// TwinCAT 3 PLC project TAMAR2MM
// ProgramVersion: 3.1.4024.0
// libraries:
//   Tc2_MC2, * (Beckhoff Automation GmbH)
//   Tc2_Standard, * (Beckhoff Automation GmbH)
//   Tc2_System, * (Beckhoff Automation GmbH)
//   Tc2_Utilities, * (Beckhoff Automation GmbH)
//   Tc3_Module, * (Beckhoff Automation GmbH)
//   VisuDialogs, * (System)
// project tree:
//   / GlobalTextList.TcGTLO, PlcTask.TcTTO (not stored), Visualization Manager.TcVMO (not stored), VISU_TASK.TcTTO (not stored)
//   POUs/AXES/ AXES_CYCLE.TcPOU, FB_Axis.TcPOU, GVL_AXES.TcGVL (not stored), vAXIS.TcVIS, vAXIS_CONTROLLER.TcVIS, AXES_SCREEN.TcVIS
//   POUs/EVENT_LOGGER/ E_EventType.TcDUT, FB_EventLogger.TcPOU, GVL_EVENT_LOGGER.TcGVL, ST_Event.TcDUT, UpdateEventTimestampWithSystemTime.TcPOU (not stored), UpdateTimeStamp.TcPOU (not stored), vEVENT_LOGGER.TcVIS (not stored)
//   POUs/ E_STATE.TcDUT, GVL_MAIN.TcGVL, MACHINE.TcPOU, MAIN.TcPOU
//   POUs/IO/ EL1809.TcDUT, EL2809.TcDUT, GVL_IO.TcGVL, ST_VTUG.TcDUT
//   POUs/PISTONS/ E_PISTON_STATE.TcDUT, E_PISTON_TYPE.TcDUT, FB_PISTON.TcPOU, GVL_PISTONS.TcGVL, PIST_CYCLE.TcPOU, ST_PISTON.TcDUT (not stored), vPISTONS.TcVIS (not stored), vPISTON.TcVIS
//   POUs/STATIONS/ FB_FEEDER.TcPOU, FB_SEPARATE.TcPOU, FB_STATION.TcPOU, STATION_CYCLE.TcPOU, vFEEDER.TcVIS, vSEPARATE.TcVIS, vSTATION_CONTROLLER.TcVIS
//   VISUs/ vCOMM.TcVIS, vMACHINE.TcVIS
// real-time tasks:
//   TASK PlcTask: cycle T#10ms, priority 20, ADS port 350
//   TASK VISU_TASK: cycle T#200000us, priority 30, ADS port 351
// motion (NC):
//   TASK NC-Task 1 SAF: cycle T#2ms, priority 4, ADS port 501
//   TASK NC-Task 1 SVB: cycle T#10ms, priority 8, ADS port 511
//   AXIS MAIN_CONV (id 1)
//     OtherSettings: AllowMotionCmdToSlave=true
//     encoder EncType=1
//     drive DrvType=5
//       Analog: TorqueSetpointScale=10, ScaleFactorActTorque=0.1
//       TimeComp: TaskDelayCycles=1
//     controller CtrType=1
//       CtrPara: PriorControlFactor=1
//         Observer: BandWidth=20
//   AXIS SUP_CONV (id 2)
//     OtherSettings: AllowMotionCmdToSlave=true
//     encoder EncType=1
//     drive DrvType=5
//       Analog: TorqueSetpointScale=10, ScaleFactorActTorque=0.1
//       TimeComp: TaskDelayCycles=1
//     controller CtrType=1
//       CtrPara: PriorControlFactor=1
//         Observer: BandWidth=20
//   AXIS PRESS1A (id 3)
//     OtherSettings: AllowMotionCmdToSlave=true
//     encoder EncType=1
//     drive DrvType=5
//       Analog: TorqueSetpointScale=10, ScaleFactorActTorque=0.1
//       TimeComp: TaskDelayCycles=1
//     controller CtrType=1
//       CtrPara: PriorControlFactor=1
//         Observer: BandWidth=20
//   AXIS PRESS1B (id 4)
//     OtherSettings: AllowMotionCmdToSlave=true
//     encoder EncType=1
//     drive DrvType=5
//       Analog: TorqueSetpointScale=10, ScaleFactorActTorque=0.1
//       TimeComp: TaskDelayCycles=1
//     controller CtrType=1
//       CtrPara: PriorControlFactor=1
//         Observer: BandWidth=20
// variable links:
//   TAMAR2MM/TAMAR2MM Instance <-> NC-Task 1 SAF/Axes/MAIN_CONV
//     PlcTask Inputs/GVL_MAIN.MAIN_CONV.Axis.NcToPlc <-> Outputs/ToPlc
//     PlcTask Outputs/GVL_MAIN.MAIN_CONV.Axis.PlcToNc <-> Inputs/FromPlc
//   TAMAR2MM/TAMAR2MM Instance <-> NC-Task 1 SAF/Axes/SUP_CONV
//     PlcTask Inputs/GVL_MAIN.SUP_CONV.Axis.NcToPlc <-> Outputs/ToPlc
//     PlcTask Outputs/GVL_MAIN.SUP_CONV.Axis.PlcToNc <-> Inputs/FromPlc

// ---- POUs/EVENT_LOGGER/E_EventType.TcDUT
{attribute 'qualified_only'}
{attribute 'strict'}
TYPE E_EventType :
(
	Alarm := 0,
	Message:=1
);
END_TYPE

// ---- POUs/EVENT_LOGGER/ST_Event.TcDUT
TYPE ST_Event :
STRUCT
	eEventType: STRING(255); 
	eEventSeverity: STRING(255);
	nEventIdentity: UDINT;
	sEventName: STRING(255);
	sEventText: STRING(255);
	dtTimestamp: DATE_AND_TIME;
	
END_STRUCT
END_TYPE

// ---- POUs/E_STATE.TcDUT
{attribute 'qualified_only'}
{attribute 'strict'}
TYPE E_STATE :
(
	uninit:=0,
	ready,
	busy,
	error
	
);
END_TYPE

// ---- POUs/IO/EL1809.TcDUT
TYPE EL1809 :
STRUCT
	ch1		:BOOL;
	ch2		:BOOL;
	ch3		:BOOL;
	ch4		:BOOL;
	ch5		:BOOL;
	ch6		:BOOL;
	ch7		:BOOL;
	ch8		:BOOL;
	ch9		:BOOL;
	ch10		:BOOL;
	ch11		:BOOL;
	ch12		:BOOL;
	ch13		:BOOL;
	ch14		:BOOL;
	ch15		:BOOL;
	ch16		:BOOL;	
END_STRUCT
END_TYPE

// ---- POUs/IO/EL2809.TcDUT
TYPE EL2809 :
STRUCT
	ch1		:BOOL;
	ch2		:BOOL;
	ch3		:BOOL;
	ch4		:BOOL;
	ch5		:BOOL;
	ch6		:BOOL;
	ch7		:BOOL;
	ch8		:BOOL;
	ch9		:BOOL;
	ch10		:BOOL;
	ch11		:BOOL;
	ch12		:BOOL;
	ch13		:BOOL;
	ch14		:BOOL;
	ch15		:BOOL;
	ch16		:BOOL;	
END_STRUCT
END_TYPE

// ---- POUs/IO/ST_VTUG.TcDUT
TYPE ST_VTUG :
STRUCT
	sol_14: BOOL;
	sol_12: BOOL;
END_STRUCT
END_TYPE

// ---- POUs/PISTONS/E_PISTON_STATE.TcDUT
{attribute 'qualified_only'}
{attribute 'strict'}
TYPE E_PISTON_STATE :
(
	uninit:=0,
	ready,
	opening,
	opened,
	closing,
	closed,
	error,
	busy
);
END_TYPE

// ---- POUs/PISTONS/E_PISTON_TYPE.TcDUT
{attribute 'qualified_only'}
{attribute 'strict'}
TYPE E_PISTON_TYPE :
(
	NO_SENSORS,
	ONLY_OPEN,
	ONLY_CLOSE,
	BOTH
);
END_TYPE

// ---- POUs/EVENT_LOGGER/GVL_EVENT_LOGGER.TcGVL
//{attribute 'qualified_only'}
VAR_GLOBAL
	// ================================== error and logs ==============================
	sError:STRING;
	gEventType: STRING(255); 
	gEventSeverity: STRING(255);
	gEventIdentity: UDINT:=0;
	gEventText: STRING(255):='Startup Event';
	gEventName: STRING(255);
	sEventTime: STRING(255);
	fbEventLogger: FB_EventLogger;
	WriteLogToFile:BOOL:=FALSE;
	sLog:STRING(255);
	bBuffer_full:BOOL:=FALSE;
END_VAR

// ---- POUs/GVL_MAIN.TcGVL
//{attribute 'qualified_only'}
VAR_GLOBAL
	fbFEEDER: FB_FEEDER;
	fbSEPARATE1: FB_SEPARATE;
	fbSEPARATE2: FB_SEPARATE;
	MAIN_CONV:FB_Axis;
	SUP_CONV:FB_Axis;
	PRESS1A:FB_Axis;
	PRESS1B:FB_Axis;
	PIST1: FB_PISTON;
	PIST2: FB_PISTON;
	
	bMAIN_HOME:BOOL:=FALSE;
	bMAIN_HOMED:BOOL:=FALSE;
	sMAIN_STATE:STRING:='UNINIT';
	eMAIN_STATE: E_STATE:=E_STATE.uninit;
	bMAIN_RESET:BOOL:=FALSE;
	iMAIN_STATE: INT:=98;
	bMAIN_PAUSE:BOOL:=FALSE;
	bMAIN_START:BOOL:=FALSE;
	
END_VAR

// ---- POUs/IO/GVL_IO.TcGVL
//{attribute 'qualified_only'}
VAR_GLOBAL
	uIOLINK1 AT%Q* : ULINT;
	uIOLINK2 AT%Q* : ULINT;	

	inputs AT %I* : ARRAY [1..4] OF EL1809;
	outputs AT %Q* : ARRAY[1..1] OF EL2809;
	
	//manifold AT %Q* : ARRAY[1..3] OF ST_VTUG;

END_VAR

// ---- POUs/PISTONS/GVL_PISTONS.TcGVL
//{attribute 'qualified_only'}
VAR_GLOBAL
	
	pFEEDER_PUSH:  FB_PISTON;
	pFEEDER_HOLD1: FB_PISTON;
	pFEEDER_HOLD2: FB_PISTON;
	pFEEDER_OPEN1: FB_PISTON;
	pFEEDER_OPEN2: FB_PISTON;
	
	pSEPARATE1_LIFT:   FB_PISTON;
	pSEPARATE1_PUSH:   FB_PISTON;
	pSEPARATE1_COLET1: FB_PISTON;
	pSEPARATE1_COLET2: FB_PISTON;
	pSEPARATE1_COLET3: FB_PISTON;
	pSEPARATE1_COLET4: FB_PISTON;
	pSEPARATE1_JACK1:  FB_PISTON;
	pSEPARATE1_JACK2:  FB_PISTON;
	pSEPARATE1_JACK3:  FB_PISTON;
	pSEPARATE1_JACK4:  FB_PISTON;
	pSEPARATE1_DRAWR:  FB_PISTON;
	pSEPARATE1_PINS1:  FB_PISTON;
	pSEPARATE1_PINS2:  FB_PISTON;
	
	pSEPARATE2_PUSH:   FB_PISTON;
	pSEPARATE2_LIFT:   FB_PISTON;
	pSEPARATE2_COLET1: FB_PISTON;
	pSEPARATE2_COLET2: FB_PISTON;
	pSEPARATE2_COLET3: FB_PISTON;
	pSEPARATE2_COLET4: FB_PISTON;
	pSEPARATE2_JACK1:  FB_PISTON;
	pSEPARATE2_JACK2:  FB_PISTON;
	pSEPARATE2_JACK3:  FB_PISTON;
	pSEPARATE2_JACK4:  FB_PISTON;
	pSEPARATE2_DRAWR:  FB_PISTON;
	pSEPARATE2_PINS1:  FB_PISTON;
	pSEPARATE2_PINS2:  FB_PISTON;
	
	
	
END_VAR

// ---- POUs/EVENT_LOGGER/FB_EventLogger.TcPOU
FUNCTION_BLOCK FB_EventLogger
VAR_INPUT
END_VAR
VAR_OUTPUT
END_VAR
VAR
	buffer_counter:INT;
	EventBuffer: ARRAY[1..MAXIMUN_SIZE_OF_EVENT_BUFFR] OF ST_Event;
	EventBuffer_clear: ARRAY[1..MAXIMUN_SIZE_OF_EVENT_BUFFR] OF ST_Event;
	EventBufferIndex:INT:=0;
END_VAR
VAR CONSTANT
	MAXIMUN_SIZE_OF_EVENT_BUFFR:INT :=100;
END_VAR

METHOD IsEventBufferFull : BOOL
VAR_INPUT
END_VAR
IF (EventBufferIndex+1) > MAXIMUN_SIZE_OF_EVENT_BUFFR THEN
	EventBuffer:=EventBuffer_clear;
	EventBufferIndex:=0 ;
	//IsEventBufferFull:=TRUE; 
END_IF
IsEventBufferFull:=FALSE;
END_METHOD

(* returns false if not succesfull*) 
METHOD PUBLIC mAdd : BOOL
VAR_INPUT
	
END_VAR

VAR
	arrDataToWrite: INT;
END_VAR

IF NOT IsEventBufferFull() THEN
	EventBufferIndex:=EventBufferIndex+1;
	EventBuffer[EventBufferIndex].eEventType:=gEventType;
	EventBuffer[EventBufferIndex].eEventSeverity:=gEventSeverity;
	EventBuffer[EventBufferIndex].nEventIdentity:=gEventIdentity;
	EventBuffer[EventBufferIndex].sEventName:=gEventName;
	EventBuffer[EventBufferIndex].sEventText:=gEventText;
	UpdateEventTimestampWithSystemTime (stEvent:=EventBuffer[EventBufferIndex]); 
	sEventTime:= DT_TO_STRING (EventBuffer[EventBufferIndex].dtTimestamp);
	mAdd:=TRUE ;
ELSE
	mAdd:=FALSE;
END_IF
END_METHOD

END_FUNCTION_BLOCK

// ---- POUs/STATIONS/FB_FEEDER.TcPOU
FUNCTION_BLOCK FB_FEEDER EXTENDS FB_STATION
VAR_INPUT
	fbPUSH: REFERENCE TO FB_PISTON;
	fbHOLD1: REFERENCE TO FB_PISTON;
	fbHOLD2: REFERENCE TO FB_PISTON;
	fbOPEN1: REFERENCE TO FB_PISTON;
	fbOPEN2: REFERENCE TO FB_PISTON;
	rACTION_TIME: TIME;
	bTEST:BOOL;
END_VAR
VAR_OUTPUT
END_VAR
VAR
	bSTART_ACTION:BOOL;
	
END_VAR

tACTION(IN:= bSTART_ACTION, PT:=rACTION_TIME , Q=> , ET=> );
IF bRESET THEN
	bRESET:=FALSE;
	iSTATION_STATE:=98 ;
	bPAUSE:=FALSE;
END_IF

IF iSTATION_STATE<>98 AND (fbHOLD1.eSTATE= E_STATE.error OR fbHOLD2.eSTATE= E_STATE.error OR fbOPEN1.eSTATE= E_STATE.error OR fbOPEN2.eSTATE= E_STATE.error OR fbPUSH.eSTATE= E_STATE.error)  THEN 
	iSTATION_STATE:=99;
END_IF

CASE iSTATION_STATE OF 
	1:
		bHOME:=FALSE;
		iSTATION_STATE:=100;
		bHOMED:=TRUE;
	2: //open open hold
		bSTART:=FALSE;
		eSTATE:=E_STATE.busy;
		sSTATION_STATE:='HOLD AND OPEN';
		fbHOLD1.aOPEN();
		fbHOLD2.aOPEN();
		fbOPEN1.aOPEN();
		fbOPEN2.aOPEN();
		IF fbHOLD1.eSTATE= E_STATE.busy AND fbHOLD2.eSTATE= E_STATE.busy AND fbOPEN1.eSTATE= E_STATE.busy AND fbOPEN2.eSTATE= E_STATE.busy  THEN
			iSTATION_STATE:=3;
		END_IF
	3://wait fo open and hold and then push
		IF  fbHOLD1.eSTATE= E_STATE.ready AND fbHOLD2.eSTATE= E_STATE.ready AND fbOPEN1.eSTATE= E_STATE.ready AND fbOPEN2.eSTATE= E_STATE.ready THEN
			IF NOT bPAUSE THEN
				sSTATION_STATE:='OPEN PUSH';
				fbPUSH.aOPEN();
				IF fbPUSH.eSTATE= E_STATE.busy THEN
					iSTATION_STATE:=4;
				END_IF
			END_IF
		END_IF
	4:	//wait for push and close push
		IF fbPUSH.eSTATE= E_STATE.ready THEN
			IF NOT bPAUSE THEN
				sSTATION_STATE:='CLOSE PUSH';
				fbPUSH.aCLOSE();
				IF fbPUSH.eSTATE= E_STATE.busy THEN
					iSTATION_STATE:=5;
				END_IF
			END_IF
		END_IF
	5://wait for push close and close hold and open
		IF fbPUSH.eSTATE= E_STATE.ready THEN
			IF NOT bPAUSE THEN
				sSTATION_STATE:='RELEASE AND CLOSE';
				fbHOLD1.aCLOSE();
				fbHOLD2.aCLOSE();
				fbOPEN1.aCLOSE();
				fbOPEN2.aCLOSE();
				IF fbPUSH.eSTATE= E_STATE.ready AND fbHOLD1.eSTATE= E_STATE.ready AND fbHOLD2.eSTATE= E_STATE.ready AND fbOPEN1.eSTATE= E_STATE.ready AND fbOPEN2.eSTATE= E_STATE.ready THEN
					 iSTATION_STATE:=6;
				END_IF
			END_IF
		END_IF

	6:	//open pist 3
		IF fbPUSH.eSTATE= E_STATE.ready AND fbHOLD1.eSTATE= E_STATE.ready AND fbHOLD2.eSTATE= E_STATE.ready AND fbOPEN1.eSTATE= E_STATE.ready AND fbOPEN2.eSTATE= E_STATE.ready THEN
			iSTATION_STATE:=100;
		END_IF
	
	
	98:
		bHOMED:=FALSE;
		eSTATE:=E_STATE.uninit;
		sSTATION_STATE:='UNINIT';
		bRESET:=FALSE;
		fbPUSH.aRESET();
		fbHOLD1.aRESET();
		fbHOLD2.aRESET();
		fbOPEN1.aRESET();
		fbOPEN2.aRESET();
		IF fbPUSH.eSTATE= E_STATE.uninit AND fbHOLD1.eSTATE= E_STATE.uninit AND fbHOLD2.eSTATE= E_STATE.uninit AND fbOPEN1.eSTATE= E_STATE.uninit AND fbOPEN2.eSTATE= E_STATE.uninit THEN
			iSTATION_STATE:=980;
		END_IF
	980: 
		IF fbPUSH.eSTATE= E_STATE.ready AND fbHOLD1.eSTATE= E_STATE.ready AND fbHOLD2.eSTATE= E_STATE.ready AND fbOPEN1.eSTATE= E_STATE.ready AND fbOPEN2.eSTATE= E_STATE.ready THEN
			IF bHOME THEN
				iSTATION_STATE:=1;
			END_IF
		END_IF
		
		//IF fbPIST1.bERROR OR fbPIST2.bERROR OR fbPIST3.bERROR THEN
		//	iSTATION_STATE:=99;
	//	END_IF
	
	99:
		eSTATE:=E_STATE.error;
		sSTATION_STATE:='PISTON ERROR';
		
	100:
		eSTATE:=E_STATE.ready;
		sSTATION_STATE:='READY';
		IF bSTART THEN
			bSTART:=FALSE;
			iSTATION_STATE:=2;
		END_IF
		
END_CASE

END_FUNCTION_BLOCK

// ---- POUs/STATIONS/FB_STATION.TcPOU
FUNCTION_BLOCK FB_STATION
VAR_INPUT
	eSTATE:E_STATE:=E_STATE.uninit;
	sSTATION_STATE:STRING:='UNINIT';
	sName:STRING;
	bHOMED : BOOL:=FALSE;
	tACTION:TON;
	bPAUSE:BOOL:=FALSE;
	bHOME: BOOL:=FALSE;
	
	
END_VAR
VAR_OUTPUT
END_VAR
VAR
	bERROR:BOOL;
	bRESET:BOOL;
	bSTART:BOOL:=FALSE;
	iSTATION_STATE:INT:=98;;
	bFIRST_RUN:BOOL:=FALSE;
END_VAR

ACTION aHOME:
bHOME:=TRUE;
END_ACTION

ACTION aRESET:
bRESET:=TRUE;
END_ACTION

ACTION aSTART:
bSTART:=TRUE;
END_ACTION

END_FUNCTION_BLOCK

// ---- POUs/PISTONS/FB_PISTON.TcPOU
FUNCTION_BLOCK FB_PISTON
VAR_INPUT
	eSTATE:E_STATE:=E_STATE.uninit;
	sSTATE:STRING:='UNINIT';
	sNAME:STRING;
	bLOCAL_MANUAL: BOOL:=FALSE;
	pist_TYPE: E_PISTON_TYPE;
	pist_STATE: E_PISTON_STATE:=E_PISTON_STATE.uninit;
	rOPEN_TIME: TIME;
	rCLOSE_TIME: TIME;
	rOPEN_TIMEOUT: TIME;
	tCLOSE_TIMEOUT: TIME;
	bOPEN_LIMIT: BOOL;
	bCLOSED_LIMIT: BOOL;
	bOPEN_CMD: BOOL;
	bCLOSE_CMD: BOOL;
	bOPEN_SWR: BOOL;
	bCLOSE_SWR: BOOL;
	bCONDITION: BOOL:=TRUE;
	bLOCAL_RESET:BOOL;
	bOPEN_DEFAULT: BOOL;
	
END_VAR
VAR_OUTPUT
	bOPEN_VALVE: BOOL;
	bCLOSE_VALVE: BOOL;
	bBUSY:BOOL;
	bOPENED:BOOL;
	bCLOSED:BOOL;
	bERROR:BOOL:=FALSE;
END_VAR
VAR
	T_OPEN: TON;
	T_OPEN_TIMEOUT: TON;
	T_CLOSE: TON;
	T_CLOSE_TIMEOUT: TON;
	
	bFIRST_DONE: BOOL:=FALSE;
	
END_VAR

T_OPEN(IN:= bOPEN_CMD, PT:=rOPEN_TIME , Q=> , ET=> );
T_CLOSE(IN:=  NOT bOPEN_CMD, PT:=rCLOSE_TIME , Q=> , ET=> );
T_OPEN_TIMEOUT(IN:= bOPEN_CMD , PT:= rOPEN_TIMEOUT, Q=> , ET=> );
T_CLOSE_TIMEOUT(IN:=  NOT bOPEN_CMD , PT:= tCLOSE_TIMEOUT, Q=> , ET=> );

IF bLOCAL_RESET THEN//========================== RESET================
	bLOCAL_RESET:=FALSE;
	pist_STATE:=E_PISTON_STATE.uninit;
END_IF

IF NOT bLOCAL_MANUAL THEN//====================== MANUAL ==============
	bOPEN_CMD:=bOPEN_SWR;
END_IF

IF NOT bFIRST_DONE THEN  // ============== check default mode ===============
	bFIRST_DONE:=TRUE;
	bOPEN_CMD:=bOPEN_DEFAULT;
END_IF
//================================================== UNINIT =====================================================
CASE pist_STATE OF
	E_PISTON_STATE.uninit:
		eSTATE:=E_STATE.uninit;
		bOPEN_CMD:=bOPEN_DEFAULT;
		bOPEN_SWR:=bOPEN_DEFAULT;
		bERROR:=FALSE;
		IF bOPEN_CMD  THEN
			bOPEN_VALVE:=TRUE;
			bCLOSE_VALVE:=FALSE;
			pist_STATE:=E_PISTON_STATE.opening;
		ELSE
			bOPEN_VALVE:=FALSE;
			bCLOSE_VALVE:=TRUE;
			pist_STATE:=E_PISTON_STATE.closing;
		END_IF
//================================================== OPENING =====================================================
	E_PISTON_STATE.opening:
	eSTATE:=E_STATE.busy;
	sSTATE:='OPENING';
	bBUSY:=TRUE; bOPENED:=FALSE; bCLOSED:=FALSE;
	CASE pist_TYPE OF//------------------------------no sensors
		E_PISTON_TYPE.NO_SENSORS:
		IF T_OPEN.Q THEN
			pist_STATE:=E_PISTON_STATE.opened;
		END_IF
		//----------------------------- both sensors
		E_PISTON_TYPE.BOTH:
		IF bOPEN_LIMIT THEN
			pist_STATE:=E_PISTON_STATE.opened;
		END_IF
		IF T_OPEN_TIMEOUT.Q THEN
			bOPEN_CMD:=FALSE;
			aPISTON_ERROR();
			pist_STATE:=E_PISTON_STATE.error;
		END_IF
		//----------------------------- only open sensor
		E_PISTON_TYPE.ONLY_OPEN:
		IF bOPEN_LIMIT THEN
			pist_STATE:=E_PISTON_STATE.opened;
		END_IF
		IF T_OPEN_TIMEOUT.Q THEN
			bOPEN_CMD:=FALSE;
			aPISTON_ERROR();
			pist_STATE:=E_PISTON_STATE.error;
		END_IF
		//----------------------------- only close sensor
		E_PISTON_TYPE.ONLY_CLOSE:
		IF T_OPEN.Q THEN
			pist_STATE:=E_PISTON_STATE.opened;
		END_IF
	END_CASE
//================================================== CLOSING =====================================================	
	E_PISTON_STATE.closing:
	eSTATE:=E_STATE.busy;
	sSTATE:='CLOSING'; bOPENED:=FALSE; bCLOSED:=FALSE;
	bBUSY:=TRUE;
	CASE pist_TYPE OF//--------------------------------------- no sensors
		E_PISTON_TYPE.NO_SENSORS:
		IF T_CLOSE.Q THEN
			pist_STATE:=E_PISTON_STATE.closed;
		END_IF
		//-------------------------------------- both sensors
		E_PISTON_TYPE.BOTH:
		IF bCLOSED_LIMIT THEN
			pist_STATE:=E_PISTON_STATE.closed;
		END_IF
		IF T_CLOSE_TIMEOUT.Q THEN
			bOPEN_CMD:=TRUE;
			pist_STATE:=E_PISTON_STATE.error;
		END_IF
		//-------------------------------------- only close sensor
		E_PISTON_TYPE.ONLY_CLOSE:
		IF bCLOSED_LIMIT THEN
			pist_STATE:=E_PISTON_STATE.closed;
		END_IF
		IF T_CLOSE_TIMEOUT.Q THEN
			bOPEN_CMD:=TRUE;
			aPISTON_ERROR();
			pist_STATE:=E_PISTON_STATE.error;
		END_IF
		//----------------------------- only close sensor
		E_PISTON_TYPE.ONLY_OPEN:
		IF T_CLOSE.Q THEN
			pist_STATE:=E_PISTON_STATE.closed;
		END_IF
	END_CASE
//================================================== OPENED =====================================================	
	E_PISTON_STATE.opened:
	eSTATE:=E_STATE.ready;
	sSTATE:='OPENED';
	bBUSY:=FALSE; bOPENED:=TRUE; bCLOSED:=FALSE;
	IF NOT bOPEN_CMD  THEN
		pist_STATE:=E_PISTON_STATE.closing;
		bOPEN_VALVE:=FALSE;
		bCLOSE_VALVE:=TRUE;
	END_IF
	CASE pist_TYPE OF
		//-------------------------------------- both sensors
		E_PISTON_TYPE.BOTH:
		IF NOT bOPEN_LIMIT THEN
			bOPEN_CMD:=FALSE;
			aPISTON_ERROR();
			pist_STATE:=E_PISTON_STATE.error;
		END_IF
		//-------------------------------------- only open sensor
		E_PISTON_TYPE.ONLY_OPEN:
		IF NOT bOPEN_LIMIT THEN
			bOPEN_CMD:=FALSE;
			aPISTON_ERROR();
			pist_STATE:=E_PISTON_STATE.error;
		END_IF
	END_CASE
//================================================== CLOSED =====================================================	
	E_PISTON_STATE.closed:
	eSTATE:=E_STATE.ready;
	sSTATE:='CLOSED';
	bBUSY:=FALSE; bOPENED:=FALSE; bCLOSED:=TRUE;
	IF bOPEN_CMD  THEN
		pist_STATE:=E_PISTON_STATE.opening;
		bOPEN_VALVE:=TRUE;
		bCLOSE_VALVE:=FALSE;
	END_IF
	CASE pist_TYPE OF
		//-------------------------------------- both sensors
		E_PISTON_TYPE.BOTH:
		IF NOT bCLOSED_LIMIT THEN
			bOPEN_CMD:=TRUE;
			aPISTON_ERROR();
			pist_STATE:=E_PISTON_STATE.error;
		END_IF
		//-------------------------------------- only close sensor
		E_PISTON_TYPE.ONLY_CLOSE:
		IF NOT bCLOSED_LIMIT THEN
			bOPEN_CMD:=TRUE;
			aPISTON_ERROR();
			pist_STATE:=E_PISTON_STATE.error;
		END_IF
	END_CASE
//================================================== ERROR =====================================================	
	E_PISTON_STATE.error:
		eSTATE:=E_STATE.error;
		sSTATE:='ERROR';
		bERROR:=TRUE;
	//
END_CASE

ACTION aCLOSE:
bOPEN_SWR:=FALSE;
END_ACTION

ACTION aHOME:
IF bOPEN_DEFAULT THEN
	bOPEN_SWR:=TRUE;
ELSE
	bOPEN_SWR:=FALSE;
END_IF
END_ACTION

ACTION aOPEN:
bOPEN_SWR:=TRUE;
END_ACTION

ACTION aPISTON_ERROR:
gEventType:= 'piston Alarm'; 
gEventSeverity:= 'Error';

gEventName:= sNAME;
IF pist_STATE=E_PISTON_STATE.opening  THEN
	gEventText:='piston opening';
	gEventIdentity:=1001;
END_IF
IF pist_STATE=E_PISTON_STATE.closing THEN
	gEventText:='piston closing';
	gEventIdentity:=1002;
END_IF
IF pist_STATE=E_PISTON_STATE.closed THEN
	gEventText:='piston closed';
	gEventIdentity:=1003;
END_IF
IF pist_STATE=E_PISTON_STATE.opened THEN
	gEventText:='piston opened';
	gEventIdentity:=1004;
END_IF
fbEventLogger.mAdd();
END_ACTION

ACTION aRESET:
bLOCAL_RESET:=TRUE;
END_ACTION

END_FUNCTION_BLOCK

// ---- POUs/STATIONS/FB_SEPARATE.TcPOU
FUNCTION_BLOCK FB_SEPARATE  EXTENDS FB_STATION
VAR_INPUT
	fbPUSH:   REFERENCE TO FB_PISTON;
	fbLIFT:   REFERENCE TO FB_PISTON;
	fbCOLET1: REFERENCE TO FB_PISTON;
	fbCOLET2: REFERENCE TO FB_PISTON;
	fbCOLET3: REFERENCE TO FB_PISTON;
	fbCOLET4: REFERENCE TO FB_PISTON;
	fbJACK1:  REFERENCE TO FB_PISTON;
	fbJACK2:  REFERENCE TO FB_PISTON;
	fbJACK3:  REFERENCE TO FB_PISTON;
	fbJACK4:  REFERENCE TO FB_PISTON;
	fbDRAWR:  REFERENCE TO FB_PISTON;
	fbPINS1:  REFERENCE TO FB_PISTON;
	fbPINS2:  REFERENCE TO FB_PISTON;
	fbPRESS1A:REFERENCE TO FB_Axis;
	fbPRESS1B:REFERENCE TO FB_Axis;
	
END_VAR
VAR_OUTPUT
END_VAR
VAR
END_VAR

IF bRESET THEN
	bRESET:=FALSE;
	iSTATION_STATE:=98 ;
	bPAUSE:=FALSE;
END_IF

IF iSTATION_STATE<>98 AND (fbLIFT.eSTATE= E_STATE.error OR
							 fbCOLET1.eSTATE= E_STATE.error OR 
								fbCOLET2.eSTATE= E_STATE.error OR
									fbCOLET3.eSTATE= E_STATE.error OR 
										fbCOLET4.eSTATE= E_STATE.error OR
											fbJACK1.eSTATE= E_STATE.error OR
												 fbJACK2.eSTATE= E_STATE.error OR 
													fbJACK3.eSTATE= E_STATE.error OR
														fbJACK4.eSTATE= E_STATE.error OR 
															fbDRAWR.eSTATE= E_STATE.error OR
																fbPINS1.eSTATE= E_STATE.error OR
												 					fbPINS2.eSTATE= E_STATE.error OR
																		fbPUSH.eSTATE= E_STATE.error  )THEN									
																										 
	iSTATION_STATE:=99;
END_IF

CASE iSTATION_STATE OF 
	1: //open pist 1
		bSTART:=FALSE;
		eSTATE:=E_STATE.busy;
		sSTATION_STATE:='LIFT DOWN';
		fbLIFT.aOPEN();
		IF fbLIFT.eSTATE= E_STATE.busy THEN
			iSTATION_STATE:=2;
		END_IF
	2://wait for LIFT ready
		IF fbLIFT.eSTATE= E_STATE.ready THEN
			IF NOT bPAUSE THEN
				iSTATION_STATE:=3;
			END_IF
		END_IF
	3:	//CLOSE COLET 1 2  ======================================= SEPARATE A =====================
		sSTATION_STATE:='CLOSE COLET 1 2';
		fbCOLET1.aOPEN();
		fbCOLET2.aOPEN();
		IF fbCOLET1.eSTATE= E_STATE.busy AND fbCOLET2.eSTATE= E_STATE.busy THEN
			iSTATION_STATE:=4;
		END_IF
	4:// WAIT FOR COLET 1 2
		IF fbCOLET1.eSTATE= E_STATE.ready AND fbCOLET2.eSTATE= E_STATE.ready THEN
			IF NOT bPAUSE THEN
				iSTATION_STATE:=5;
			END_IF
		END_IF
	5:	//SEPARATE A 
		sSTATION_STATE:='SEPARATE A';
		fbLIFT.aCLOSE();
		fbPRESS1A.mMOVE_REL(1000);
		fbPRESS1B.mMOVE_REL(1000);
		
		IF fbLIFT.eSTATE= E_STATE.busy AND fbPRESS1A.eSTATE= E_STATE.busy AND fbPRESS1B.eSTATE= E_STATE.busy THEN
			iSTATION_STATE:=6;
		END_IF
	6:
		IF  fbPRESS1A.eSTATE= E_STATE.ready AND fbPRESS1B.eSTATE= E_STATE.ready THEN
			IF NOT bPAUSE THEN
				iSTATION_STATE:=7;
			END_IF
		END_IF
		
	7:	//CLOSE COLET 1 2  ======================================= SEPARATE B =====================
		sSTATION_STATE:='CLOSE COLET 3 4';
		fbCOLET3.aOPEN();
		fbCOLET4.aOPEN();
		IF fbCOLET3.eSTATE= E_STATE.busy AND fbCOLET4.eSTATE= E_STATE.busy THEN
			iSTATION_STATE:=8;
		END_IF
	8:// WAIT FOR COLET 1 2
		IF fbCOLET3.eSTATE= E_STATE.ready AND fbCOLET4.eSTATE= E_STATE.ready THEN
			IF NOT bPAUSE THEN
				iSTATION_STATE:=9;
			END_IF
		END_IF
	9:	//SEPARATE A 
		sSTATION_STATE:='SEPARATE B';
		fbPRESS1A.mMOVE_REL(1000);
		fbPRESS1B.mMOVE_REL(1000);
		
		IF fbPRESS1A.eSTATE= E_STATE.busy AND fbPRESS1B.eSTATE= E_STATE.busy THEN
			iSTATION_STATE:=10;
		END_IF
	10:
		IF  fbLIFT.eSTATE= E_STATE.ready AND fbPRESS1A.eSTATE= E_STATE.ready AND fbPRESS1B.eSTATE= E_STATE.ready THEN
			IF NOT bPAUSE THEN
				iSTATION_STATE:=11;
			END_IF
		END_IF
		
		//========================================================================== CLEARING =======================
	11:	
		sSTATION_STATE:='OPEN DRAWER';
		fbDRAWR.aOPEN();
		IF fbDRAWR.eSTATE= E_STATE.busy  THEN
			iSTATION_STATE:=12;
		END_IF
	12:
		IF fbDRAWR.eSTATE= E_STATE.ready THEN
			IF NOT bPAUSE THEN
				iSTATION_STATE:=13;
			END_IF
		END_IF
	13:	//open colets
		sSTATION_STATE:='OPEN COLETS';
		fbCOLET1.aCLOSE();
		fbCOLET2.aCLOSE();
		fbCOLET3.aCLOSE();
		fbCOLET4.aCLOSE();
		IF fbCOLET1.eSTATE= E_STATE.busy AND fbCOLET2.eSTATE= E_STATE.busy AND fbCOLET3.eSTATE= E_STATE.busy AND fbCOLET4.eSTATE= E_STATE.busy THEN
			iSTATION_STATE:=14;
		END_IF
	14:
		IF fbCOLET1.eSTATE= E_STATE.ready AND fbCOLET2.eSTATE= E_STATE.ready AND fbCOLET3.eSTATE= E_STATE.ready AND fbCOLET4.eSTATE= E_STATE.ready THEN
			IF NOT bPAUSE THEN
				iSTATION_STATE:=15;
			END_IF
		END_IF	
	15:	//press pins
		sSTATION_STATE:='PINS OUT';
		fbPINS1.aOPEN();
		fbPINS2.aOPEN();
		IF fbPINS1.eSTATE= E_STATE.busy AND fbPINS2.eSTATE= E_STATE.busy THEN
			iSTATION_STATE:=16;
		END_IF
	16:
		IF fbPINS1.eSTATE= E_STATE.ready AND fbPINS2.eSTATE= E_STATE.ready THEN
			IF NOT bPAUSE THEN
				iSTATION_STATE:=17;
			END_IF
		END_IF
	17:	//pins up and push
		sSTATION_STATE:='PINS UP AND PUSH';
		fbPINS1.aCLOSE();
		fbPINS2.aCLOSE();
		fbPUSH.aOPEN();
		IF fbPUSH.eSTATE= E_STATE.busy AND fbPINS1.eSTATE= E_STATE.busy AND fbPINS2.eSTATE= E_STATE.busy THEN
			iSTATION_STATE:=18;
		END_IF
	18:
		IF  fbPUSH.eSTATE= E_STATE.ready AND fbPINS1.eSTATE= E_STATE.ready AND fbPINS2.eSTATE= E_STATE.ready THEN
			IF NOT bPAUSE THEN
				iSTATION_STATE:=19;
			END_IF
		END_IF
	19:	//close drawer jacks down
		sSTATION_STATE:='CLOSE DRAWER JACKS DOWN';
		fbDRAWR.aCLOSE();
		fbPRESS1A.aHOME();
		fbPRESS1B.aHOME();
		IF fbDRAWR.eSTATE= E_STATE.busy AND fbPRESS1A.eSTATE= E_STATE.busy AND fbPRESS1B.eSTATE= E_STATE.busy THEN
			iSTATION_STATE:=20;
		END_IF
	20:
		IF  fbLIFT.eSTATE= E_STATE.ready AND fbDRAWR.eSTATE= E_STATE.ready AND fbPRESS1A.bHOME AND fbPRESS1B.bHOMED THEN
			IF NOT bPAUSE THEN
				iSTATION_STATE:=100;
			END_IF
		END_IF

	
	98:
		eSTATE:=E_STATE.uninit;
		sSTATION_STATE:='UNINIT';
		bRESET:=FALSE;
		fbPRESS1A.aHOME();
		fbPRESS1B.aHOME();
		fbPUSH.aRESET();
		fbLIFT.aRESET();
		fbCOLET1.aRESET();
		fbCOLET2.aRESET();
		fbCOLET3.aRESET();
		fbCOLET4.aRESET();
		fbJACK1.aRESET();
		fbJACK2.aRESET();
		fbJACK3.aRESET();
		fbJACK4.aRESET();
		fbDRAWR.aRESET();
		fbPINS1.aRESET();
		fbPINS2.aRESET();
		
		IF fbPRESS1A.eSTATE= E_STATE.busy AND 
					fbPRESS1B.eSTATE= E_STATE.busy AND 
						fbLIFT.eSTATE= E_STATE.uninit AND
							 fbCOLET1.eSTATE= E_STATE.uninit AND
								fbCOLET2.eSTATE= E_STATE.uninit AND
									fbCOLET3.eSTATE= E_STATE.uninit AND
										fbCOLET4.eSTATE= E_STATE.uninit AND
											fbJACK1.eSTATE= E_STATE.uninit AND
												 fbJACK2.eSTATE= E_STATE.uninit AND 
													fbJACK3.eSTATE= E_STATE.uninit AND
														fbJACK4.eSTATE= E_STATE.uninit AND 
															fbDRAWR.eSTATE= E_STATE.uninit AND
																fbPINS1.eSTATE= E_STATE.uninit AND
												 					fbPINS2.eSTATE= E_STATE.uninit AND
																		fbPUSH.eSTATE= E_STATE.uninit THEN
			iSTATION_STATE:=980;
		END_IF
	980: 
		IF fbPRESS1A.bHOMED AND 
				fbPRESS1B.bHOMED AND 
					fbLIFT.eSTATE= E_STATE.ready AND
						 fbCOLET1.eSTATE= E_STATE.ready AND
							fbCOLET2.eSTATE= E_STATE.ready AND
								fbCOLET3.eSTATE= E_STATE.ready AND
									fbCOLET4.eSTATE= E_STATE.ready AND
										fbJACK1.eSTATE= E_STATE.ready AND
											fbJACK2.eSTATE= E_STATE.ready AND 
												fbJACK3.eSTATE= E_STATE.ready AND
													fbJACK4.eSTATE= E_STATE.ready AND 
														fbDRAWR.eSTATE= E_STATE.ready AND
															fbPINS1.eSTATE= E_STATE.ready AND
																fbPINS2.eSTATE= E_STATE.ready AND
																	fbPUSH.eSTATE= E_STATE.ready THEN
			iSTATION_STATE:=100;
		END_IF
		
	
	99:
		eSTATE:=E_STATE.error;
		sSTATION_STATE:='ERROR';
		
	100:
		eSTATE:=E_STATE.ready;
		sSTATION_STATE:='READY';
		IF bSTART THEN
			bSTART:=FALSE;
			iSTATION_STATE:=1;
		END_IF
		
END_CASE

END_FUNCTION_BLOCK

// ---- POUs/AXES/FB_Axis.TcPOU
FUNCTION_BLOCK FB_Axis
VAR_INPUT
	eSTATE:E_STATE:=E_STATE.uninit;
	sAXIS_STATE:STRING:='UNINIT';
	sName:STRING;
	Axis:Axis_ref;
	bEnable:BOOL:=FALSE;
	bHalt:BOOL:=FALSE;
	bHOME:BOOL:=FALSE;
	bHOME_DIR:BOOL;
	bReset:BOOL:=FALSE;
	bSetPosition:BOOL:=FALSE;
	Dist:REAL;
	bMoveRel:BOOL:=FALSE;
	bMoveRelBusy:BOOL;
	rPos:LREAL;
	rVel:LREAL;
	rAcc:LREAL;
	rDec:LREAL;
	rJerk:LREAL;
	bMoveABS:BOOL:=FALSE;
	bMoveAbsBusy:BOOL;
	bJogPos:BOOL;
	bJogNeg:BOOL;
	bMANUAL:BOOL:=FALSE;
	tACTION:TON;
	ton_Reset: TON;
	bOPEN:BOOL;
	bCLOSE:BOOL;
	bLIMIT_OPENED:BOOL;
	bLIMIT_CLOSED:BOOL;
	bLIMIT:BOOL;
	rACTION_TIMEOUT:TIME:=T#10S;
	jogVEL: REAL;
	bSTOP:BOOL;
	SKIP_HOME :BOOL:=TRUE;
END_VAR

VAR_OUTPUT
	bOPENED:BOOL;
	bCLOSED:BOOL;
	bHOMED:BOOL;
	bBusy: BOOL;
	bAXIS_ERROR:BOOL;
	bSTATE_ERROR:BOOL;
	bInPos:BOOL;
	rActPos:LREAL;
	rActVel:LREAL;
	bRelDone:BOOL;
	bAbsDone:BOOL;
	bHaltDone:BOOL;
END_VAR
VAR
	bSTART_ACTION:BOOL;
	iHOME_STATE: INT:=98;
	iAXIS_STATE:INT:=98;
	tDelay: TON;
	bDelay:BOOL:=FALSE;
	MoveAbsolute: MC_MoveAbsolute;
	power: MC_Power;
	Reset: MC_Reset;
	SetPosition: MC_SetPosition;
	JOG: MC_Jog;
	RELATIVE: MC_MoveRelative;
	HALT: MC_Halt;
	HOME: MC_Home;
	bFirst_run:BOOL:=FALSE;
	bStopBusy:BOOL;
	
	
	
	
END_VAR

IF NOT bFirst_run THEN
	RESET.Execute:=TRUE;
	 bFirst_run:=TRUE;
END_IF

rActPos:=Axis.NcToPlc.ActPos;
rActVel:=Axis.NcToPlc.ActVelo;

IF RELATIVE.Done AND bMoveRel THEN
	bMoveRel:=FALSE;
END_IF

IF MoveAbsolute.Done AND bMoveAbs THEN
	bMoveAbs:=FALSE;
END_IF

IF RELATIVE.Busy OR JOG.Busy OR moveAbsolute.busy  THEN
	bBusy:=TRUE;
	//bInpos:=FALSE;
END_IF

IF NOT RELATIVE.Busy AND NOT JOG.Busy AND NOT moveAbsolute.busy  THEN
	bBusy:=FALSE;
	//bInpos:=TRUE;
END_IF

IF POWER.error OR RELATIVE.error OR MoveAbsolute.error OR JOG.error THEN
	bAXIS_ERROR:=TRUE;
END_IF


IF bRelDone OR  bAbsDone THEN
	bInPos:=TRUE;
END_IF


IF bBusy THEN
	bInPos:=FALSE;
	bRelDone:=FALSE;
	bAbsDone:=FALSE;
END_IF


CMDs();
mAXIS_STATE_MACHINE();

ACTION aAXIS_ERROR:
gEventType:= 'axis Alarm'; 
gEventSeverity:= 'Error';

gEventName:= sNAME;
IF iAXIS_STATE=1  THEN
	gEventText:='axis homing';
	gEventIdentity:=2001;
END_IF
IF iAXIS_STATE=20  THEN
	gEventText:='axis opening';
	gEventIdentity:=2002;
END_IF
IF iAXIS_STATE=40  THEN
	gEventText:='axis closing';
	gEventIdentity:=2003;
END_IF
fbEventLogger.mAdd();
END_ACTION

ACTION aHOME:
bHOME:=TRUE;
END_ACTION

ACTION aRESET:
iAXIS_STATE:=98;
bHOME:=FALSE;
END_ACTION

METHOD clear_cmd_req : BOOL
VAR_INPUT
END_VAR

bMoveABS:= bMoveRel:= bJogPos:= bJogNeg:=FALSE;
END_METHOD

ACTION CMDs:
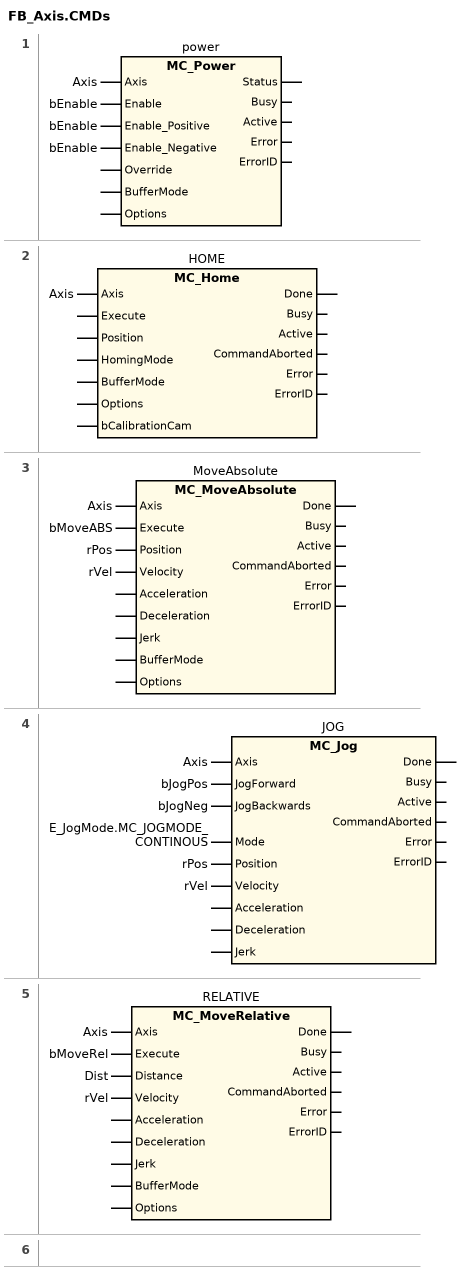
// NETWORK 1
power(Axis := Axis, Enable := bEnable, Enable_Positive := bEnable, Enable_Negative := bEnable); // MC_Power

// NETWORK 2
HOME(Axis := Axis); // MC_Home

// NETWORK 3
MoveAbsolute(Axis := Axis, Execute := bMoveABS, Position := rPos, Velocity := rVel); // MC_MoveAbsolute

// NETWORK 4
JOG(
    Axis := Axis,
    JogForward := bJogPos,
    JogBackwards := bJogNeg,
    Mode := E_JogMode.MC_JOGMODE_CONTINOUS,
    Position := rPos,
    Velocity := rVel); // MC_Jog

// NETWORK 5
RELATIVE(Axis := Axis, Execute := bMoveRel, Distance := Dist, Velocity := rVel); // MC_MoveRelative

// NETWORK 6

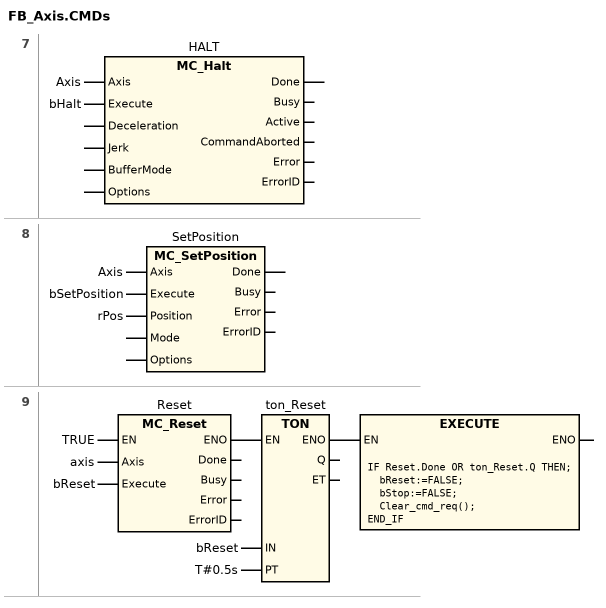
// NETWORK 7
HALT(Axis := Axis, Execute := bHalt); // MC_Halt

// NETWORK 8
SetPosition(Axis := Axis, Execute := bSetPosition, Position := rPos); // MC_SetPosition

// NETWORK 9
Reset(Axis := axis, Execute := bReset); // MC_Reset
ton_Reset(IN := bReset, PT := T#0.5s); // TON

IF Reset.Done OR ton_Reset.Q THEN;
	bReset:=FALSE;
	bStop:=FALSE;
	Clear_cmd_req();
END_IF
END_ACTION

METHOD mAXIS_STATE_MACHINE : BOOL
VAR_INPUT
	
END_VAR
tACTION(IN:= bSTART_ACTION, PT:=rACTION_TIMEOUT , Q=> , ET=> );
IF bHOME_DIR THEN
	bLIMIT:=bLIMIT_OPENED;
ELSE
	bLIMIT:=bLIMIT_CLOSED;
END_IF


CASE iAXIS_STATE OF
	1:// ============================================== HOMING
		bENABLE:=TRUE;
		bHOME:=FALSE;
		IF SKIP_HOME THEN
			bHOMED:=TRUE;
			IF bHOME_DIR THEN
				iAXIS_STATE:=100;// to ready state
			ELSE
				iAXIS_STATE:=100;// to ready state
			END_IF
		ELSE
			eSTATE:=E_STATE.busy;
			bSTART_ACTION:=TRUE;
			sAXIS_STATE:='HOMING - TO SENSOR';
			bHOMED:=FALSE;bHOME:=FALSE;
			bENABLE:=TRUE;
			rVel:= jogVEL;
			IF bHOME_DIR THEN
				bJogPos:=TRUE;
			ELSE
				bJogNeg:=TRUE;
			END_IF
			
			IF bLIMIT THEN
				bSTART_ACTION:=FALSE;
				bJogNeg:=FALSE;
				bJogPos:=FALSE;
				iAXIS_STATE:=2;
			END_IF
			IF tACTION.Q THEN
				bSTART_ACTION:=FALSE;
				aAXIS_ERROR();
				iAXIS_STATE:=99;
				bSTATE_ERROR:=TRUE;
			END_IF
		END_IF
		
	2://FROM LIMIT
			sAXIS_STATE:= 'HOMING- FROM SENSOR';
			IF Axis.NcToPlc.ActVelo= 0 THEN
				rVel:= jogVEL/5;
				IF bHOME_DIR THEN
					bJogNeg:=TRUE;
				ELSE
					bJogPos:=TRUE;
				END_IF
				iAXIS_STATE:=3;
			END_IF	
	3:// FINISH
			IF NOT bLIMIT THEN
				bJogNeg:=FALSE;
				bJogPos:=FALSE;
				IF Axis.NcToPlc.ActVelo= 0 THEN
					bHOMED:=TRUE;
					IF bHOME_DIR THEN
						iAXIS_STATE:=100;// to ready state
					ELSE
						iAXIS_STATE:=100;// to ready state
					END_IF
				END_IF
			END_IF
	
	50:	//========================ABSOLUTE=====================
	eSTATE:=E_STATE.busy;
	sAXIS_STATE:='MOVING ABSOLUTE';
	bAbsDone:=FALSE; bHOMED:=FALSE;bHOME:=FALSE;
	IF moveAbsolute.Done OR HALT.Done THEN
		iAXIS_STATE:=100;
		bAbsDone:=TRUE;
		bMoveAbs:=FALSE;
	END_IF
	51://========================RELATIVE=====================
	eSTATE:=E_STATE.busy;
	sAXIS_STATE:='MOVING RELATIVE';
	bRelDone:=FALSE;bHOMED:=FALSE;bHOME:=FALSE;
	IF RELATIVE.Done OR HALT.Done THEN
		iAXIS_STATE:=100; 
		bRelDone:=TRUE;
		bMoveRel:=FALSE;
	END_IF
	52://======================= HALT =========================
	sAXIS_STATE:='HALTING';
	bHaltDone:=FALSE;bHOMED:=FALSE;bHOME:=FALSE;
	IF HALT.Done THEN
		iAXIS_STATE:=100;
		bHaltDone:=TRUE;
		bHALT:=FALSE;
	END_IF		
	98:// ====================== UNINIT =========================
		eSTATE:=E_STATE.uninit;
		sAXIS_STATE:='UNINIT';
		bENABLE:=FALSE;
		bHOMED:=FALSE;
		IF bHOME THEN
			iAXIS_STATE:=1;
			bSTATE_ERROR:=FALSE;
		END_IF
		
	99://====================== ERROR ============================
		eSTATE:=E_STATE.error;
		sAXIS_STATE:='AXIS STATE ERROR';
		bJogNeg:=FALSE;
		bJogPos:=FALSE;
		bHOMED:=FALSE;
		IF bHOME THEN
			iAXIS_STATE:=1;
			bSTATE_ERROR:=FALSE;
		END_IF
		
	100://==================== READY =============================
		eSTATE:=E_STATE.ready;
		sAXIS_STATE:='READY';
		IF bHOME AND NOT bHOMED THEN
			iAXIS_STATE:=1;
			//bSTATE_ERROR:=FALSE;
		END_IF
		IF bCLOSE AND NOT bCLOSED THEN
			iAXIS_STATE:=40;
			bSTATE_ERROR:=FALSE;
		END_IF
		IF bOPEN AND NOT bOPENED THEN
			iAXIS_STATE:=20;
			bSTATE_ERROR:=FALSE;
		END_IF
		IF bMoveAbs THEN
			bENABLE:=TRUE;
			iAXIS_STATE:=50;
			bSTATE_ERROR:=FALSE;
		END_IF
		IF bMoveRel THEN
			bENABLE:=TRUE;
			iAXIS_STATE:=51;
			bSTATE_ERROR:=FALSE;
		END_IF
		IF bHALT THEN
			iAXIS_STATE:=52;
			bSTATE_ERROR:=FALSE;
		END_IF
	
END_CASE
END_METHOD

METHOD mMOVE_ABS : BOOL
VAR_INPUT
	movement:REAL;
END_VAR
rPOS:=movement;
bMoveAbs:=TRUE;
END_METHOD

METHOD mMOVE_REL : BOOL
VAR_INPUT
	movement:REAL;
END_VAR

IF eSTATE= E_STATE.ready THEN
	Dist:=movement;
	bMoveRel:=TRUE;
END_IF
END_METHOD

END_FUNCTION_BLOCK

// ---- POUs/AXES/AXES_CYCLE.TcPOU
PROGRAM AXES_CYCLE
VAR
END_VAR

GRP1();

ACTION GRP1:
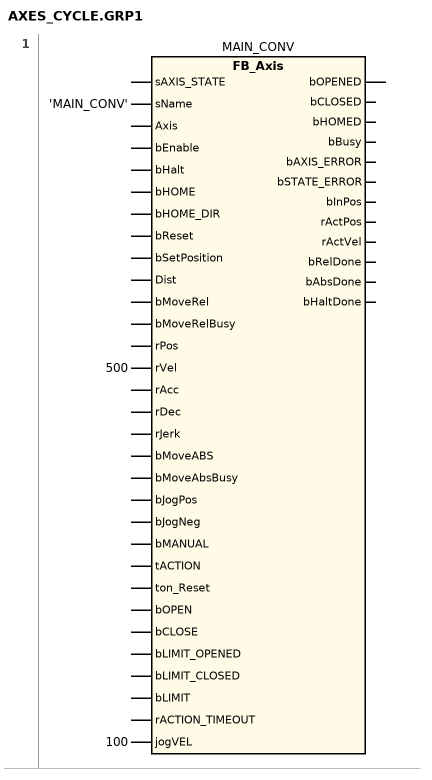
// NETWORK 1
MAIN_CONV(sName := 'MAIN_CONV', rVel := 500, jogVEL := 100); // FB_Axis

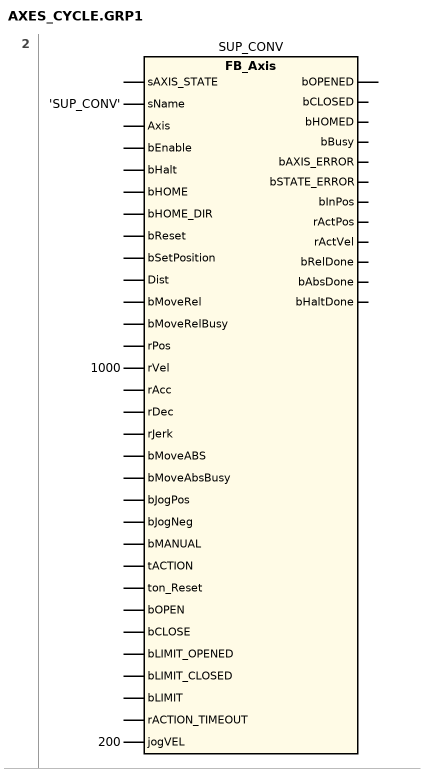
// NETWORK 2
SUP_CONV(sName := 'SUP_CONV', rVel := 1000, jogVEL := 200); // FB_Axis

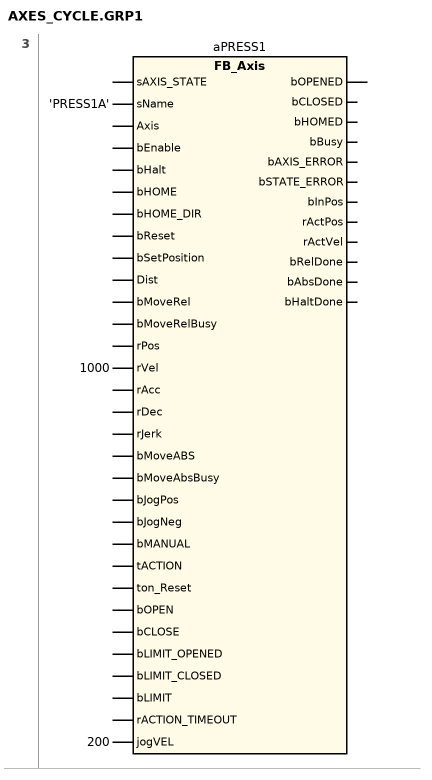
// NETWORK 3
aPRESS1(sName := 'PRESS1A', rVel := 1000, jogVEL := 200); // FB_Axis

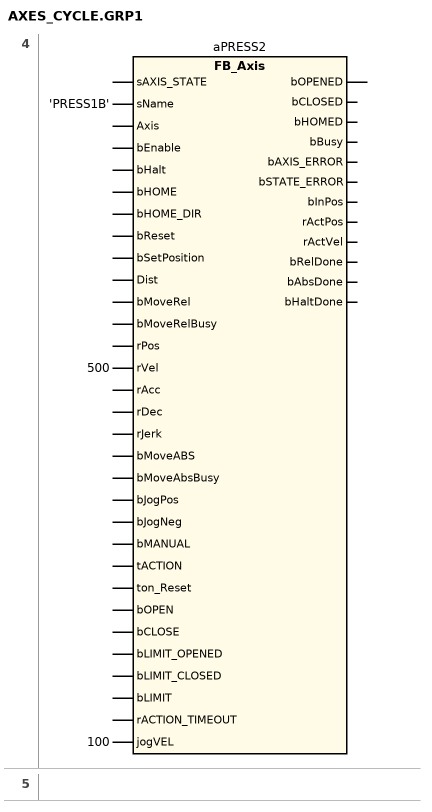
// NETWORK 4
aPRESS2(sName := 'PRESS1B', rVel := 500, jogVEL := 100); // FB_Axis

// NETWORK 5
END_ACTION

END_PROGRAM

// ---- POUs/MACHINE.TcPOU
PROGRAM MACHINE
VAR
END_VAR

IF fbFEEDER.eSTATE= E_STATE.error OR fbSEPARATE1.eSTATE= E_STATE.error OR MAIN_CONV.eSTATE= E_STATE.error OR SUP_CONV.eSTATE= E_STATE.error THEN
	iMAIN_STATE:=99 ;
END_IF

IF bMAIN_RESET THEN
	iMAIN_STATE:=98 ;
	bMAIN_PAUSE:=FALSE;
	sMAIN_STATE:='UNINIT';
END_IF

CASE iMAIN_STATE OF 
	1://===================================== HOME ============================
		MAIN_CONV.aHOME();
		SUP_CONV.aHOME();
		
		eMAIN_STATE:=E_STATE.busy;
		bMAIN_HOME:=FALSE;
		sMAIN_STATE:='HOMING';
		IF MAIN_CONV.bHOMED AND SUP_CONV.bHOMED THEN
			iMAIN_STATE:=100;
			bMAIN_HOMED:=TRUE;
		END_IF
	2: //====================================  START ==============================
		eMAIN_STATE:=E_STATE.busy;
		sMAIN_STATE:='CONVAYORS';
		MAIN_CONV.mMOVE_REL(1000);
		SUP_CONV.mMOVE_REL(1000);
		IF SUP_CONV.eSTATE= E_STATE.busy AND MAIN_CONV.eSTATE = E_STATE.busy THEN
			iMAIN_STATE:=3;
		END_IF
	3://wait for convayors
		IF SUP_CONV.eSTATE= E_STATE.ready AND MAIN_CONV.eSTATE = E_STATE.ready THEN
			IF NOT bMAIN_PAUSE THEN
				iMAIN_STATE:=4;
			END_IF
		END_IF
		
	4: //stations
		eMAIN_STATE:=E_STATE.busy;
		sMAIN_STATE:=' STANIONS';
		fbFEEDER.aSTART();
		fbSEPARATE1.aSTART();
		fbSEPARATE2.aSTART();
		IF fbSEPARATE1.eSTATE= E_STATE.busy AND fbSEPARATE2.eSTATE= E_STATE.busy AND fbFEEDER.eSTATE= E_STATE.busy THEN
			iMAIN_STATE:=5;
		END_IF
	5://wait for separate1
		IF fbSEPARATE1.eSTATE= E_STATE.ready AND fbSEPARATE2.eSTATE= E_STATE.ready AND fbFEEDER.eSTATE= E_STATE.ready THEN
			IF NOT bMAIN_PAUSE THEN
				iMAIN_STATE:=100;
			END_IF
		END_IF
		
	98://======================================== UNINIT ============================
		bMAIN_HOMED:=FALSE;
		eMAIN_STATE:=E_STATE.uninit;
		sMAIN_STATE:='UNINIT';
		bMAIN_RESET:=FALSE;
		fbFEEDER.aRESET();
		fbSEPARATE1.aRESET();
		MAIN_CONV.aRESET();
		
		IF fbFEEDER.eSTATE = E_STATE.uninit AND fbSEPARATE1.eSTATE = E_STATE.uninit AND MAIN_CONV.eSTATE=E_STATE.uninit  AND SUP_CONV.eSTATE=E_STATE.uninit THEN
			iMAIN_STATE:=980;
		END_IF
	980: 
		IF fbFEEDER.eSTATE= E_STATE.ready AND fbSEPARATE1.eSTATE= E_STATE.ready AND MAIN_CONV.eSTATE=E_STATE.uninit  AND SUP_CONV.eSTATE=E_STATE.uninit THEN
			IF bMAIN_HOME THEN
				iMAIN_STATE:=1;
			END_IF
		END_IF
	
	99://========================================== ERROR ================================
		eMAIN_STATE:=E_STATE.error;
		sMAIN_STATE:='MACHINE ERROR';
		
	100://========================================= READY ================================
		eMAIN_STATE:=E_STATE.ready;
		sMAIN_STATE:='READY';
		IF bMAIN_START THEN
			bMAIN_START:=FALSE;
			iMAIN_STATE:=2;
		END_IF
		
END_CASE

END_PROGRAM

// ---- POUs/MAIN.TcPOU
PROGRAM MAIN
VAR
	
END_VAR



AXES_CYCLE();
PIST_CYCLE();
STATION_CYCLE();
MACHINE();

END_PROGRAM

// ---- POUs/PISTONS/PIST_CYCLE.TcPOU
PROGRAM PIST_CYCLE
VAR
	bFirstRun:BOOL:=FALSE;
	counter :INT;
END_VAR


grp_feeder();
grp_separate1();
grp_separate2();

ACTION grp_feeder:
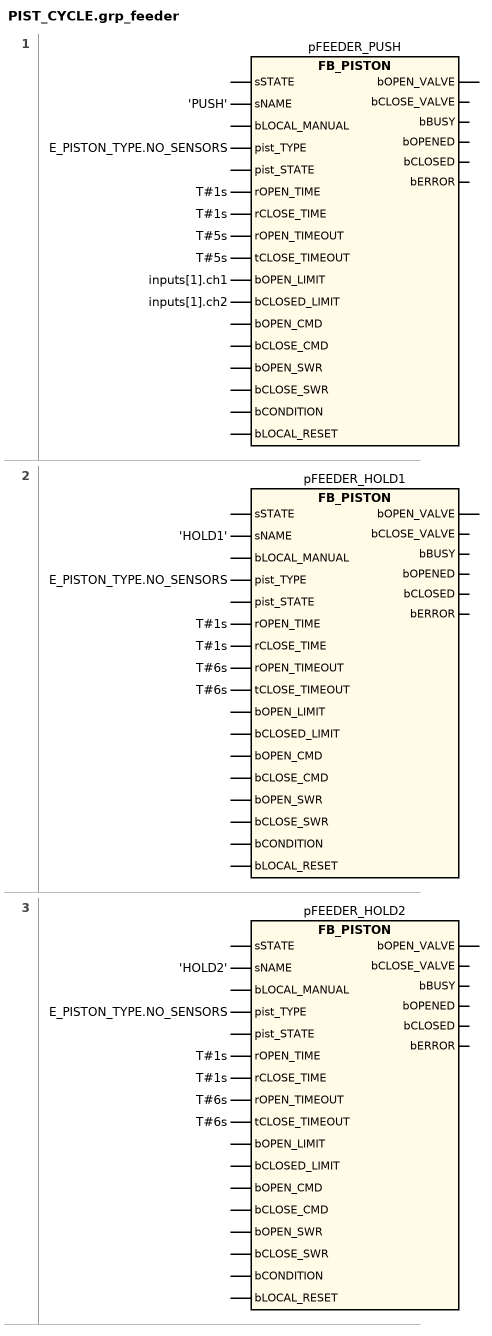
// NETWORK 1
pFEEDER_PUSH(
    sNAME := 'PUSH',
    pist_TYPE := E_PISTON_TYPE.NO_SENSORS,
    rOPEN_TIME := T#1s,
    rCLOSE_TIME := T#1s,
    rOPEN_TIMEOUT := T#5s,
    tCLOSE_TIMEOUT := T#5s,
    bOPEN_LIMIT := inputs[1].ch1,
    bCLOSED_LIMIT := inputs[1].ch2); // FB_PISTON

// NETWORK 2
pFEEDER_HOLD1(
    sNAME := 'HOLD1',
    pist_TYPE := E_PISTON_TYPE.NO_SENSORS,
    rOPEN_TIME := T#1s,
    rCLOSE_TIME := T#1s,
    rOPEN_TIMEOUT := T#6s,
    tCLOSE_TIMEOUT := T#6s); // FB_PISTON

// NETWORK 3
pFEEDER_HOLD2(
    sNAME := 'HOLD2',
    pist_TYPE := E_PISTON_TYPE.NO_SENSORS,
    rOPEN_TIME := T#1s,
    rCLOSE_TIME := T#1s,
    rOPEN_TIMEOUT := T#6s,
    tCLOSE_TIMEOUT := T#6s); // FB_PISTON

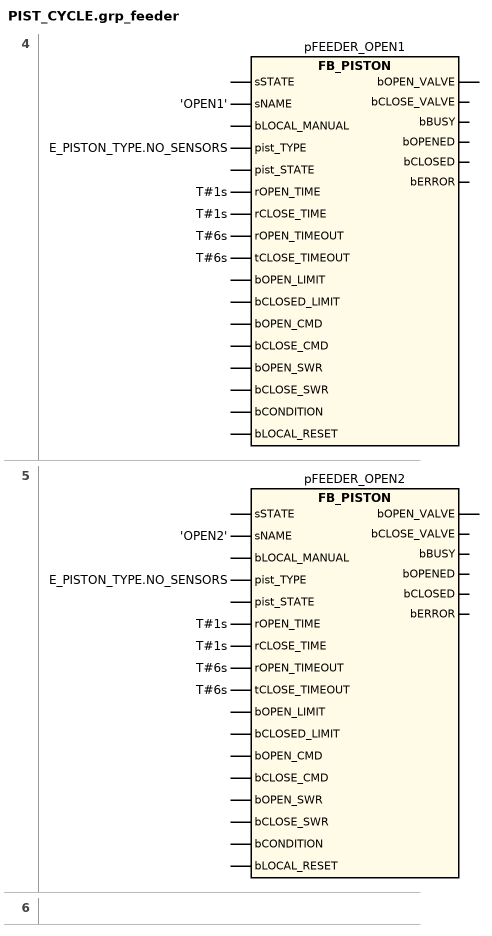
// NETWORK 4
pFEEDER_OPEN1(
    sNAME := 'OPEN1',
    pist_TYPE := E_PISTON_TYPE.NO_SENSORS,
    rOPEN_TIME := T#1s,
    rCLOSE_TIME := T#1s,
    rOPEN_TIMEOUT := T#6s,
    tCLOSE_TIMEOUT := T#6s); // FB_PISTON

// NETWORK 5
pFEEDER_OPEN2(
    sNAME := 'OPEN2',
    pist_TYPE := E_PISTON_TYPE.NO_SENSORS,
    rOPEN_TIME := T#1s,
    rCLOSE_TIME := T#1s,
    rOPEN_TIMEOUT := T#6s,
    tCLOSE_TIMEOUT := T#6s); // FB_PISTON

// NETWORK 6
END_ACTION

ACTION grp_separate1:
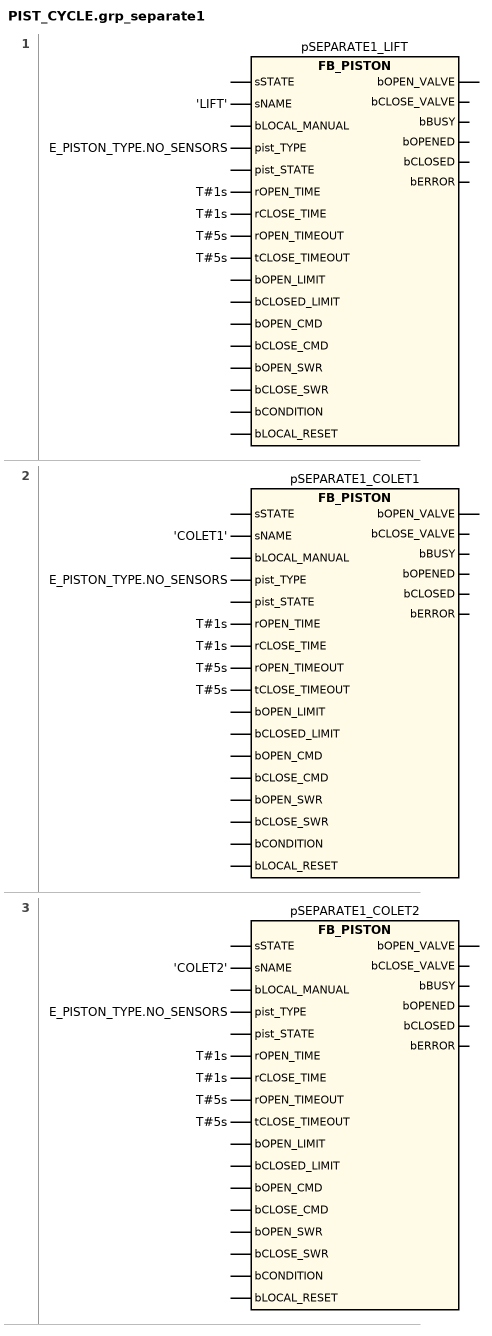
// NETWORK 1
pSEPARATE1_LIFT(
    sNAME := 'LIFT',
    pist_TYPE := E_PISTON_TYPE.NO_SENSORS,
    rOPEN_TIME := T#1s,
    rCLOSE_TIME := T#1s,
    rOPEN_TIMEOUT := T#5s,
    tCLOSE_TIMEOUT := T#5s); // FB_PISTON

// NETWORK 2
pSEPARATE1_COLET1(
    sNAME := 'COLET1',
    pist_TYPE := E_PISTON_TYPE.NO_SENSORS,
    rOPEN_TIME := T#1s,
    rCLOSE_TIME := T#1s,
    rOPEN_TIMEOUT := T#5s,
    tCLOSE_TIMEOUT := T#5s); // FB_PISTON

// NETWORK 3
pSEPARATE1_COLET2(
    sNAME := 'COLET2',
    pist_TYPE := E_PISTON_TYPE.NO_SENSORS,
    rOPEN_TIME := T#1s,
    rCLOSE_TIME := T#1s,
    rOPEN_TIMEOUT := T#5s,
    tCLOSE_TIMEOUT := T#5s); // FB_PISTON

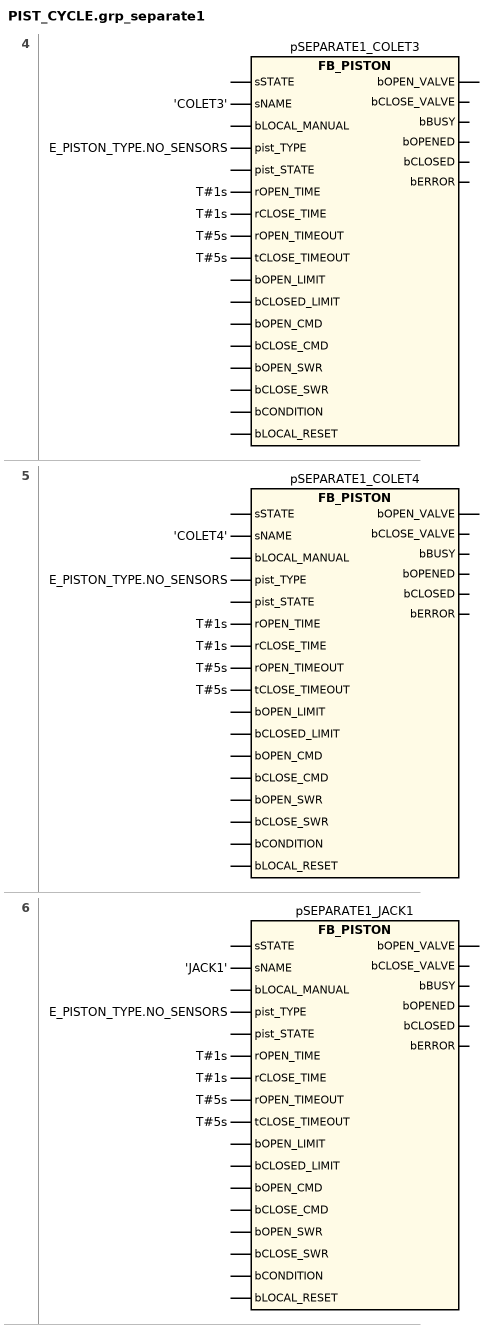
// NETWORK 4
pSEPARATE1_COLET3(
    sNAME := 'COLET3',
    pist_TYPE := E_PISTON_TYPE.NO_SENSORS,
    rOPEN_TIME := T#1s,
    rCLOSE_TIME := T#1s,
    rOPEN_TIMEOUT := T#5s,
    tCLOSE_TIMEOUT := T#5s); // FB_PISTON

// NETWORK 5
pSEPARATE1_COLET4(
    sNAME := 'COLET4',
    pist_TYPE := E_PISTON_TYPE.NO_SENSORS,
    rOPEN_TIME := T#1s,
    rCLOSE_TIME := T#1s,
    rOPEN_TIMEOUT := T#5s,
    tCLOSE_TIMEOUT := T#5s); // FB_PISTON

// NETWORK 6
pSEPARATE1_JACK1(
    sNAME := 'JACK1',
    pist_TYPE := E_PISTON_TYPE.NO_SENSORS,
    rOPEN_TIME := T#1s,
    rCLOSE_TIME := T#1s,
    rOPEN_TIMEOUT := T#5s,
    tCLOSE_TIMEOUT := T#5s); // FB_PISTON

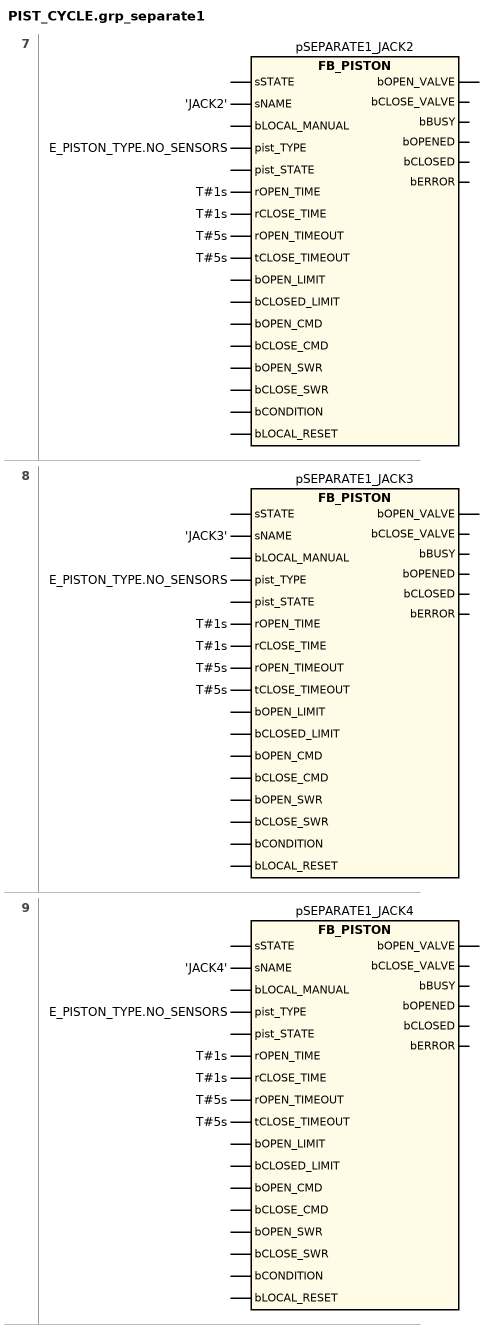
// NETWORK 7
pSEPARATE1_JACK2(
    sNAME := 'JACK2',
    pist_TYPE := E_PISTON_TYPE.NO_SENSORS,
    rOPEN_TIME := T#1s,
    rCLOSE_TIME := T#1s,
    rOPEN_TIMEOUT := T#5s,
    tCLOSE_TIMEOUT := T#5s); // FB_PISTON

// NETWORK 8
pSEPARATE1_JACK3(
    sNAME := 'JACK3',
    pist_TYPE := E_PISTON_TYPE.NO_SENSORS,
    rOPEN_TIME := T#1s,
    rCLOSE_TIME := T#1s,
    rOPEN_TIMEOUT := T#5s,
    tCLOSE_TIMEOUT := T#5s); // FB_PISTON

// NETWORK 9
pSEPARATE1_JACK4(
    sNAME := 'JACK4',
    pist_TYPE := E_PISTON_TYPE.NO_SENSORS,
    rOPEN_TIME := T#1s,
    rCLOSE_TIME := T#1s,
    rOPEN_TIMEOUT := T#5s,
    tCLOSE_TIMEOUT := T#5s); // FB_PISTON

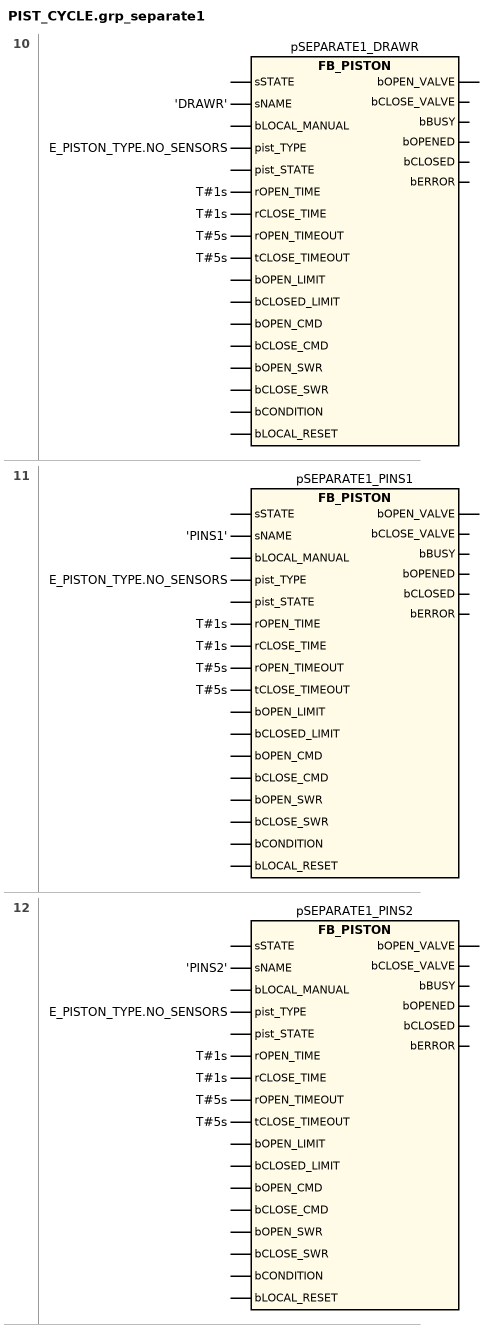
// NETWORK 10
pSEPARATE1_DRAWR(
    sNAME := 'DRAWR',
    pist_TYPE := E_PISTON_TYPE.NO_SENSORS,
    rOPEN_TIME := T#1s,
    rCLOSE_TIME := T#1s,
    rOPEN_TIMEOUT := T#5s,
    tCLOSE_TIMEOUT := T#5s); // FB_PISTON

// NETWORK 11
pSEPARATE1_PINS1(
    sNAME := 'PINS1',
    pist_TYPE := E_PISTON_TYPE.NO_SENSORS,
    rOPEN_TIME := T#1s,
    rCLOSE_TIME := T#1s,
    rOPEN_TIMEOUT := T#5s,
    tCLOSE_TIMEOUT := T#5s); // FB_PISTON

// NETWORK 12
pSEPARATE1_PINS2(
    sNAME := 'PINS2',
    pist_TYPE := E_PISTON_TYPE.NO_SENSORS,
    rOPEN_TIME := T#1s,
    rCLOSE_TIME := T#1s,
    rOPEN_TIMEOUT := T#5s,
    tCLOSE_TIMEOUT := T#5s); // FB_PISTON

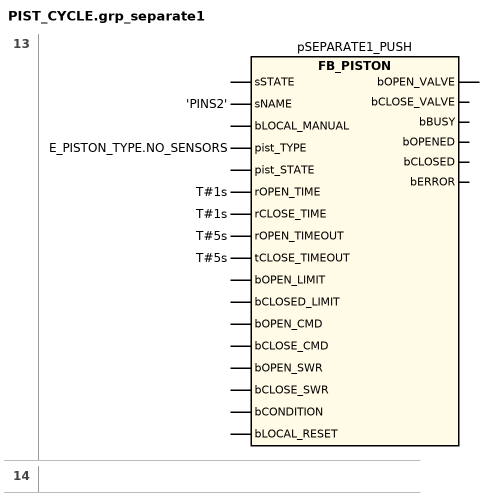
// NETWORK 13
pSEPARATE1_PUSH(
    sNAME := 'PINS2',
    pist_TYPE := E_PISTON_TYPE.NO_SENSORS,
    rOPEN_TIME := T#1s,
    rCLOSE_TIME := T#1s,
    rOPEN_TIMEOUT := T#5s,
    tCLOSE_TIMEOUT := T#5s); // FB_PISTON

// NETWORK 14
END_ACTION

ACTION grp_separate2:
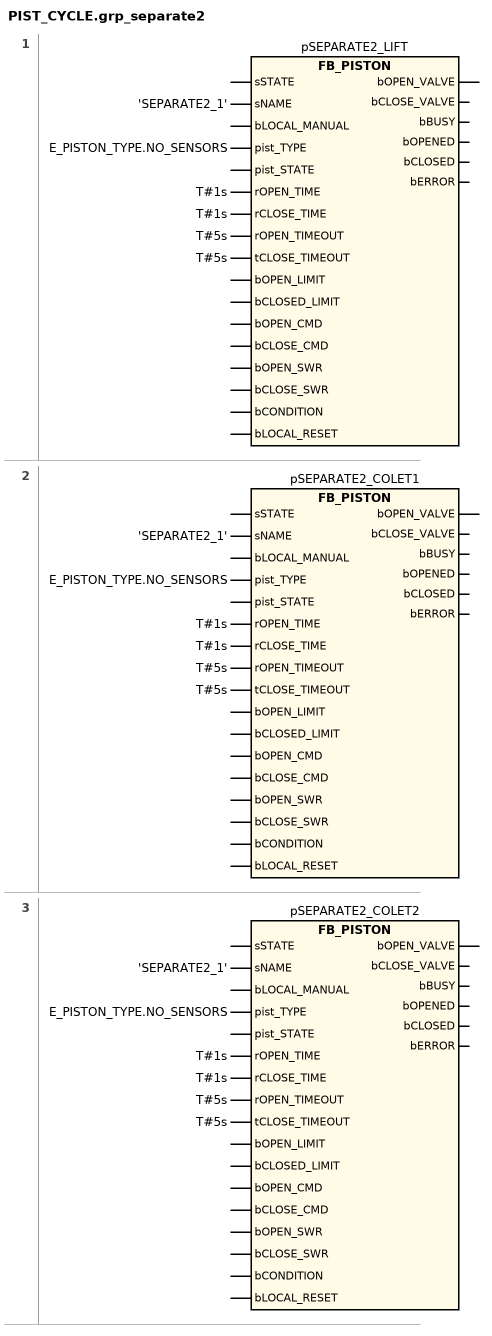
// NETWORK 1
pSEPARATE2_LIFT(
    sNAME := 'SEPARATE2_1',
    pist_TYPE := E_PISTON_TYPE.NO_SENSORS,
    rOPEN_TIME := T#1s,
    rCLOSE_TIME := T#1s,
    rOPEN_TIMEOUT := T#5s,
    tCLOSE_TIMEOUT := T#5s); // FB_PISTON

// NETWORK 2
pSEPARATE2_COLET1(
    sNAME := 'SEPARATE2_1',
    pist_TYPE := E_PISTON_TYPE.NO_SENSORS,
    rOPEN_TIME := T#1s,
    rCLOSE_TIME := T#1s,
    rOPEN_TIMEOUT := T#5s,
    tCLOSE_TIMEOUT := T#5s); // FB_PISTON

// NETWORK 3
pSEPARATE2_COLET2(
    sNAME := 'SEPARATE2_1',
    pist_TYPE := E_PISTON_TYPE.NO_SENSORS,
    rOPEN_TIME := T#1s,
    rCLOSE_TIME := T#1s,
    rOPEN_TIMEOUT := T#5s,
    tCLOSE_TIMEOUT := T#5s); // FB_PISTON

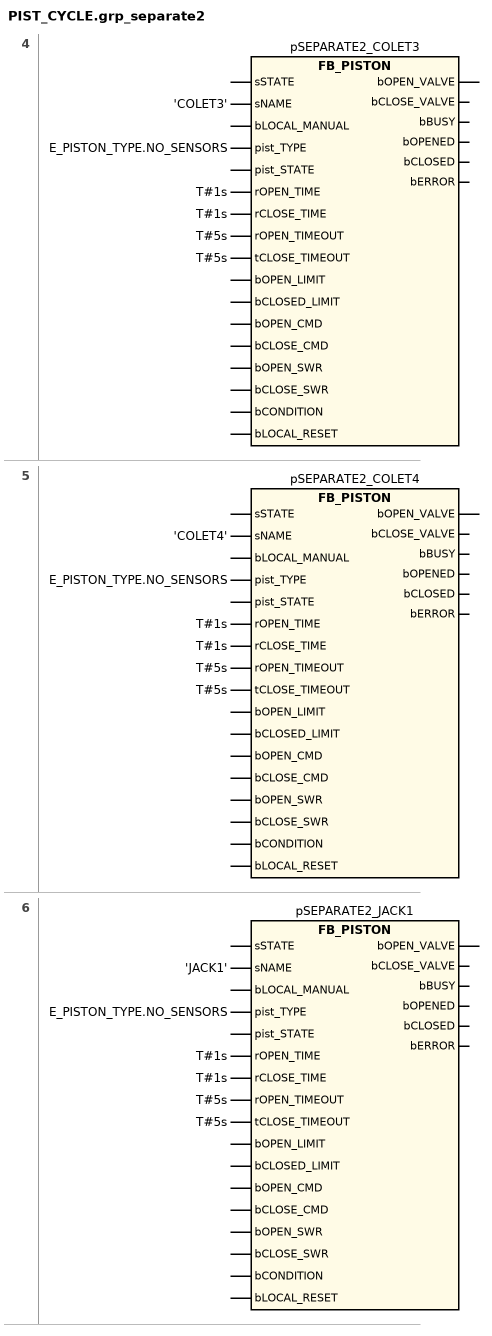
// NETWORK 4
pSEPARATE2_COLET3(
    sNAME := 'COLET3',
    pist_TYPE := E_PISTON_TYPE.NO_SENSORS,
    rOPEN_TIME := T#1s,
    rCLOSE_TIME := T#1s,
    rOPEN_TIMEOUT := T#5s,
    tCLOSE_TIMEOUT := T#5s); // FB_PISTON

// NETWORK 5
pSEPARATE2_COLET4(
    sNAME := 'COLET4',
    pist_TYPE := E_PISTON_TYPE.NO_SENSORS,
    rOPEN_TIME := T#1s,
    rCLOSE_TIME := T#1s,
    rOPEN_TIMEOUT := T#5s,
    tCLOSE_TIMEOUT := T#5s); // FB_PISTON

// NETWORK 6
pSEPARATE2_JACK1(
    sNAME := 'JACK1',
    pist_TYPE := E_PISTON_TYPE.NO_SENSORS,
    rOPEN_TIME := T#1s,
    rCLOSE_TIME := T#1s,
    rOPEN_TIMEOUT := T#5s,
    tCLOSE_TIMEOUT := T#5s); // FB_PISTON

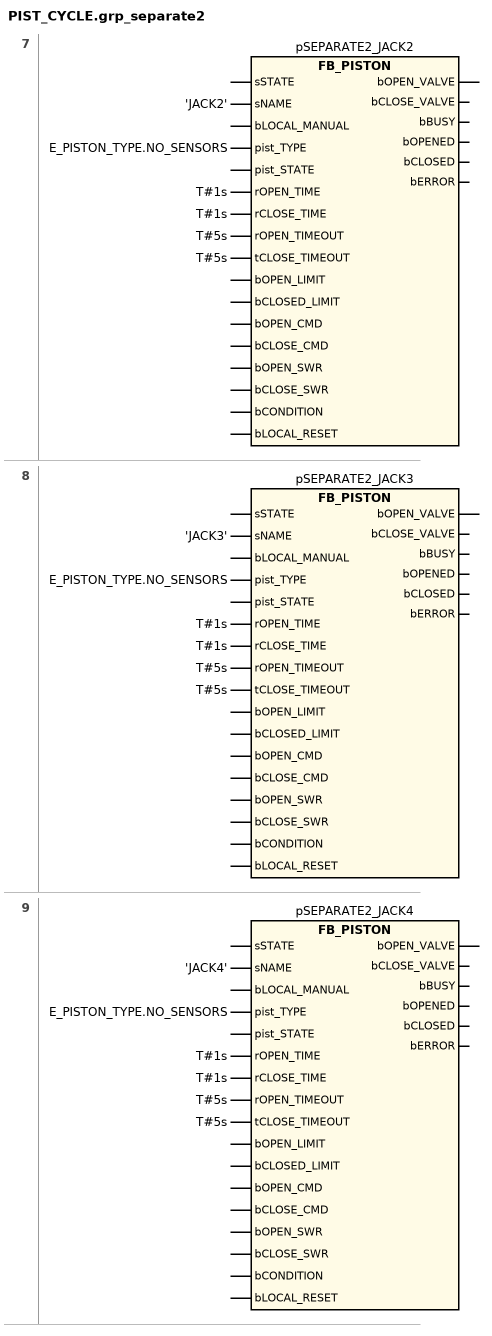
// NETWORK 7
pSEPARATE2_JACK2(
    sNAME := 'JACK2',
    pist_TYPE := E_PISTON_TYPE.NO_SENSORS,
    rOPEN_TIME := T#1s,
    rCLOSE_TIME := T#1s,
    rOPEN_TIMEOUT := T#5s,
    tCLOSE_TIMEOUT := T#5s); // FB_PISTON

// NETWORK 8
pSEPARATE2_JACK3(
    sNAME := 'JACK3',
    pist_TYPE := E_PISTON_TYPE.NO_SENSORS,
    rOPEN_TIME := T#1s,
    rCLOSE_TIME := T#1s,
    rOPEN_TIMEOUT := T#5s,
    tCLOSE_TIMEOUT := T#5s); // FB_PISTON

// NETWORK 9
pSEPARATE2_JACK4(
    sNAME := 'JACK4',
    pist_TYPE := E_PISTON_TYPE.NO_SENSORS,
    rOPEN_TIME := T#1s,
    rCLOSE_TIME := T#1s,
    rOPEN_TIMEOUT := T#5s,
    tCLOSE_TIMEOUT := T#5s); // FB_PISTON

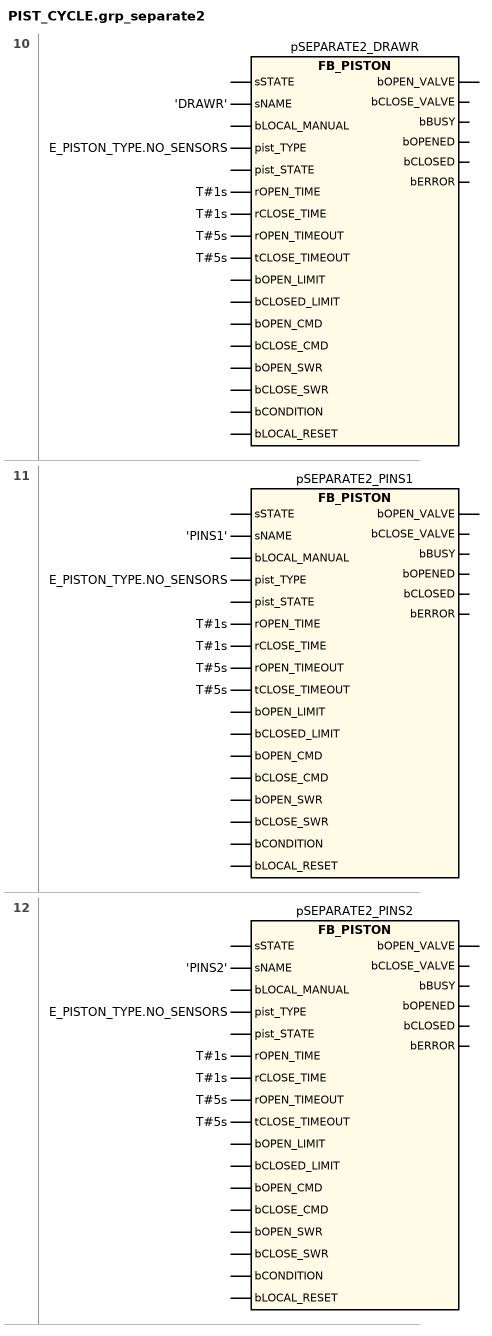
// NETWORK 10
pSEPARATE2_DRAWR(
    sNAME := 'DRAWR',
    pist_TYPE := E_PISTON_TYPE.NO_SENSORS,
    rOPEN_TIME := T#1s,
    rCLOSE_TIME := T#1s,
    rOPEN_TIMEOUT := T#5s,
    tCLOSE_TIMEOUT := T#5s); // FB_PISTON

// NETWORK 11
pSEPARATE2_PINS1(
    sNAME := 'PINS1',
    pist_TYPE := E_PISTON_TYPE.NO_SENSORS,
    rOPEN_TIME := T#1s,
    rCLOSE_TIME := T#1s,
    rOPEN_TIMEOUT := T#5s,
    tCLOSE_TIMEOUT := T#5s); // FB_PISTON

// NETWORK 12
pSEPARATE2_PINS2(
    sNAME := 'PINS2',
    pist_TYPE := E_PISTON_TYPE.NO_SENSORS,
    rOPEN_TIME := T#1s,
    rCLOSE_TIME := T#1s,
    rOPEN_TIMEOUT := T#5s,
    tCLOSE_TIMEOUT := T#5s); // FB_PISTON

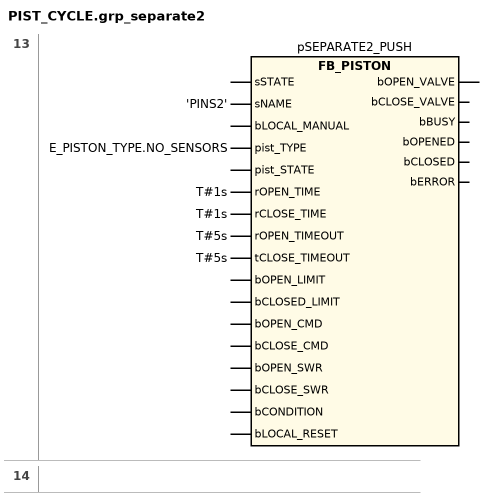
// NETWORK 13
pSEPARATE2_PUSH(
    sNAME := 'PINS2',
    pist_TYPE := E_PISTON_TYPE.NO_SENSORS,
    rOPEN_TIME := T#1s,
    rCLOSE_TIME := T#1s,
    rOPEN_TIMEOUT := T#5s,
    tCLOSE_TIMEOUT := T#5s); // FB_PISTON

// NETWORK 14
END_ACTION

END_PROGRAM

// ---- POUs/STATIONS/STATION_CYCLE.TcPOU
PROGRAM STATION_CYCLE
VAR
END_VAR

grp_feeder();
grp_separate();

ACTION grp_feeder:
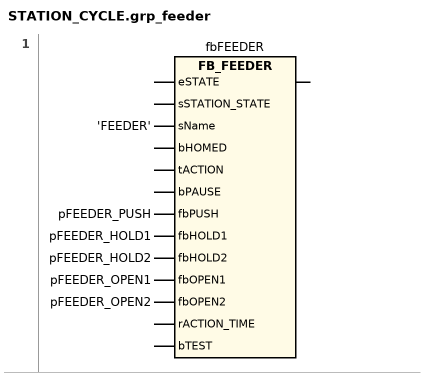
// NETWORK 1
fbFEEDER(
    sName := 'FEEDER',
    fbPUSH := pFEEDER_PUSH,
    fbHOLD1 := pFEEDER_HOLD1,
    fbHOLD2 := pFEEDER_HOLD2,
    fbOPEN1 := pFEEDER_OPEN1,
    fbOPEN2 := pFEEDER_OPEN2); // FB_FEEDER
END_ACTION

ACTION grp_separate:
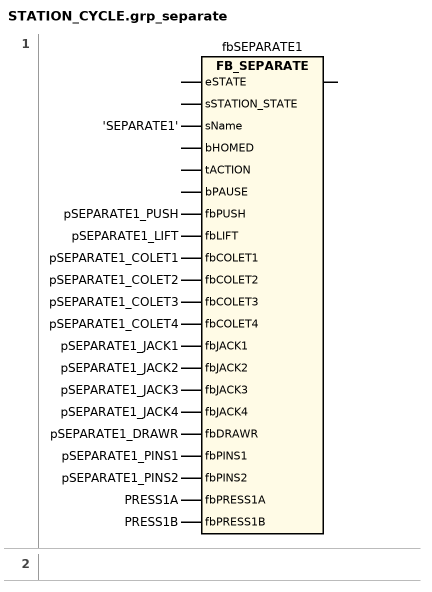
// NETWORK 1
fbSEPARATE1(
    sName := 'SEPARATE1',
    fbPUSH := pSEPARATE1_PUSH,
    fbLIFT := pSEPARATE1_LIFT,
    fbCOLET1 := pSEPARATE1_COLET1,
    fbCOLET2 := pSEPARATE1_COLET2,
    fbCOLET3 := pSEPARATE1_COLET3,
    fbCOLET4 := pSEPARATE1_COLET4,
    fbJACK1 := pSEPARATE1_JACK1,
    fbJACK2 := pSEPARATE1_JACK2,
    fbJACK3 := pSEPARATE1_JACK3,
    fbJACK4 := pSEPARATE1_JACK4,
    fbDRAWR := pSEPARATE1_DRAWR,
    fbPINS1 := pSEPARATE1_PINS1,
    fbPINS2 := pSEPARATE1_PINS2,
    fbPRESS1A := PRESS1A,
    fbPRESS1B := PRESS1B); // FB_SEPARATE

// NETWORK 2
END_ACTION

END_PROGRAM

// ---- GlobalTextList.TcGTLO
TEXTLIST GlobalTextList
  450 = '%.2f'
  859 = '%d'
  952 = '%s'
  396 = 'ACC'
  684 = 'AXES'
  188 = 'BUSY'
  997 = 'CLOSE'
  513 = 'CLOSE ALL'
  293 = 'CLOSED LIMIT'
  446 = 'DIST'
  904 = 'ENABLE'
  50 = 'ERROR'
  182 = 'ESTOP'
  810 = 'FEEDER'
  288 = 'GO ABS'
  776 = 'GO REL'
  373 = 'HALT'
  598 = 'HOME'
  566 = 'HOME ALL'
  825 = 'HOME_ALL'
  512 = 'INPOS'
  837 = 'JERK'
  268 = 'JOG +'
  202 = 'JOG -'
  309 = 'MACHINE'
  412 = 'MANUAL'
  189 = 'OPEN'
  149 = 'OPEN ALL'
  299 = 'OPENED LIMIT'
  569 = 'PAUSE'
  282 = 'PAUSED:'
  425 = 'POS'
  400 = 'POS:'
  390 = 'Pos: %.2f'
  563 = 'POWER'
  793 = 'POWER BY STRIX'
  507 = 'R'
  779 = 'RESET'
  403 = 'SEPARATE'
  917 = 'SEPARATE 1'
  71 = 'SEPARATE 2'
  830 = 'SET'
  487 = 'START'
  792 = 'STEP +'
  405 = 'STEP -'
  659 = 'STEP+'
  506 = 'STRIX1200'
  245 = 'TAMAR 20MM'
  964 = 'VEL'
  60 = 'Vel: %.2f'
END_TEXTLIST

// ---- POUs/AXES/vAXIS.TcVIS
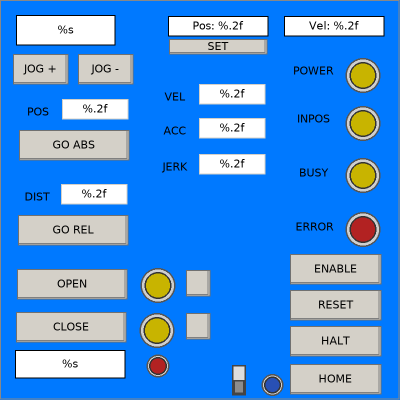
VISUALIZATION vAXIS  // 400x400
VAR_IN_OUT
	vAxis:FB_Axis;
END_VAR
    Rectangle (168,16 100x20), "Pos: %.2f", text variable: vAxis.rActPos
    Rectangle (284,16 100x20), "Vel: %.2f", text variable: vAxis.rActVel
    Lamp1 (343,53 40x45), variable: vAxis.power.Enable, style: Lamp-Lamp1-Yellow
    Label (286,60 55x22), "POWER"
    Lamp1 (343,101 40x45), variable: vAxis.bInPos, style: Lamp-Lamp1-Yellow
    Lamp1 (343,207 40x45), variable: vAxis.bAXIS_ERROR, style: Lamp-Lamp1-Red
    Lamp1 (343,153 40x45), variable: vAxis.bBusy, style: Lamp-Lamp1-Yellow
    Label (286,108 55x22), "INPOS"
    Label (287,216 55x22), "ERROR"
    Label (286,162 55x22), "BUSY"
    Button (290,254 91x30), "ENABLE"
        toggle vAxis.bEnable
    Button (290,290 91x30), "RESET"
        OnMouseDown: execute { vAXIS.bReset:=TRUE; }
    Button (290,326 91x30), "HALT"
        tap vAxis.bHalt
    Textfield (199,84 66x20), "%.2f", text variable: vAxis.rVel
        OnMouseDown: write the text variable via Default
    Label (157,86 36x22), "VEL"
    Textfield (62,99 66x20), "%.2f", text variable: vAxis.rPos
        OnMouseDown: write the text variable via Default
    Label (20,101 36x22), "POS"
    Textfield (199,154 66x20), "%.2f", text variable: vAxis.rJerk
        OnMouseDown: write the text variable via Default
    Label (157,156 36x22), "JERK"
    Textfield (199,118 66x20), "%.2f", text variable: vAxis.rAcc
        OnMouseDown: write the text variable via Default
    Label (157,120 36x22), "ACC"
    Button (13,54 55x30), "JOG +"
        tap vAxis.bJogPos
    Button (78,54 55x30), "JOG -"
        tap vAxis.bJogNeg
    Button (19,130 110x30), "GO ABS"
        OnMouseDown: execute { vAXIS.bMoveABS:=TRUE; }
    Textfield (61,184 66x20), "%.2f", text variable: vAxis.Dist
        OnMouseDown: write the text variable via Default
    Label (19,186 36x22), "DIST"
    Button (18,215 110x30), "GO REL"
        OnMouseDown: execute { vAXIS.bMoveRel:=TRUE; }
    Rectangle (16,15 99x30), "%s", text variable: vAxis.sName
    Button (169,39 98x15), "SET"
        tap vAxis.bSetPosition
    Button (17,269 110x30), "OPEN"
        OnMouseDown: execute { vAXIS.bOPEN:=TRUE;  vAXIS.bCLOSE:=FALSE; }
    Button (16,312 110x30), "CLOSE"
        OnMouseDown: execute { vAXIS.bCLOSE:=TRUE; vAXIS.bOPEN:=FALSE; }
    Lamp1 (138,263 40x45), variable: vAxis.bLIMIT_OPENED, style: Lamp-Lamp1-Yellow
    Lamp1 (137,308 40x45), variable: vAxis.bLIMIT_CLOSED, style: Lamp-Lamp1-Yellow
    Rectangle (15,350 110x28), "%s", text variable: vAxis.sAXIS_STATE
    Button (186,270 24x26)
        toggle vAxis.bLIMIT_OPENED
    Button (186,313 24x26)
        toggle vAxis.bLIMIT_CLOSED
    Button (290,364 91x30), "HOME"
        OnMouseDown: execute { vAxis.bHOME:=TRUE; }
    DipSwitch (224,365 30x30), variable: vAxis.bHOME_DIR, behaviour: TOGGLE, style: Switch-DipSwitch-Gray
    Lamp1 (260,368 25x34), variable: vAxis.bHOMED, style: Lamp-Lamp1-Blue
    Lamp1 (145,352 26x28), variable: vAxis.bSTATE_ERROR, style: Lamp-Lamp1-Red
END_VISUALIZATION

// ---- POUs/AXES/vAXIS_CONTROLLER.TcVIS
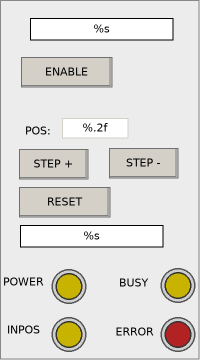
VISUALIZATION vAXIS_CONTROLLER  // 200x360
VAR_IN_OUT
	vAXIS:FB_Axis;
END_VAR
    Rectangle (30,18 143x22), "%s", text variable: vAXIS.sName
    Lamp1 (49,264 40x45), variable: vAxis.power.Enable, style: Lamp-Lamp1-Yellow
    Label (-4,271 55x22), "POWER"
    Lamp1 (49,312 40x45), variable: vAxis.bInPos, style: Lamp-Lamp1-Yellow
    Lamp1 (158,312 40x45), variable: vAxis.bAXIS_ERROR, style: Lamp-Lamp1-Red
    Lamp1 (158,263 40x45), variable: vAxis.bBusy, style: Lamp-Lamp1-Yellow
    Label (-4,319 55x22), "INPOS"
    Label (107,321 55x22), "ERROR"
    Label (106,272 55x22), "BUSY"
    Textfield (62,118 66x20), "%.2f", text variable: vAXIS.Axis.NcToPlc.ActPos
        OnMouseDown: write the text variable via Default
    Label (20,120 36x22), "POS:"
    Button (19,149 69x30), "STEP +"
        OnMouseDown: execute { vAXIS.mMOVE_REL(1000); }
    Button (21,57 91x30), "ENABLE"
        toggle vAxis.bEnable
    Button (19,187 91x30), "RESET"
        OnMouseDown: execute { vAXIS.bReset:=TRUE; }
    Button (109,148 69x30), "STEP -"
        OnMouseDown: execute { vAXIS.mMOVE_REL(-1000); }
    Rectangle (20,225 143x22), "%s", text variable: vAXIS.sAXIS_STATE
END_VISUALIZATION

// ---- POUs/AXES/AXES_SCREEN.TcVIS
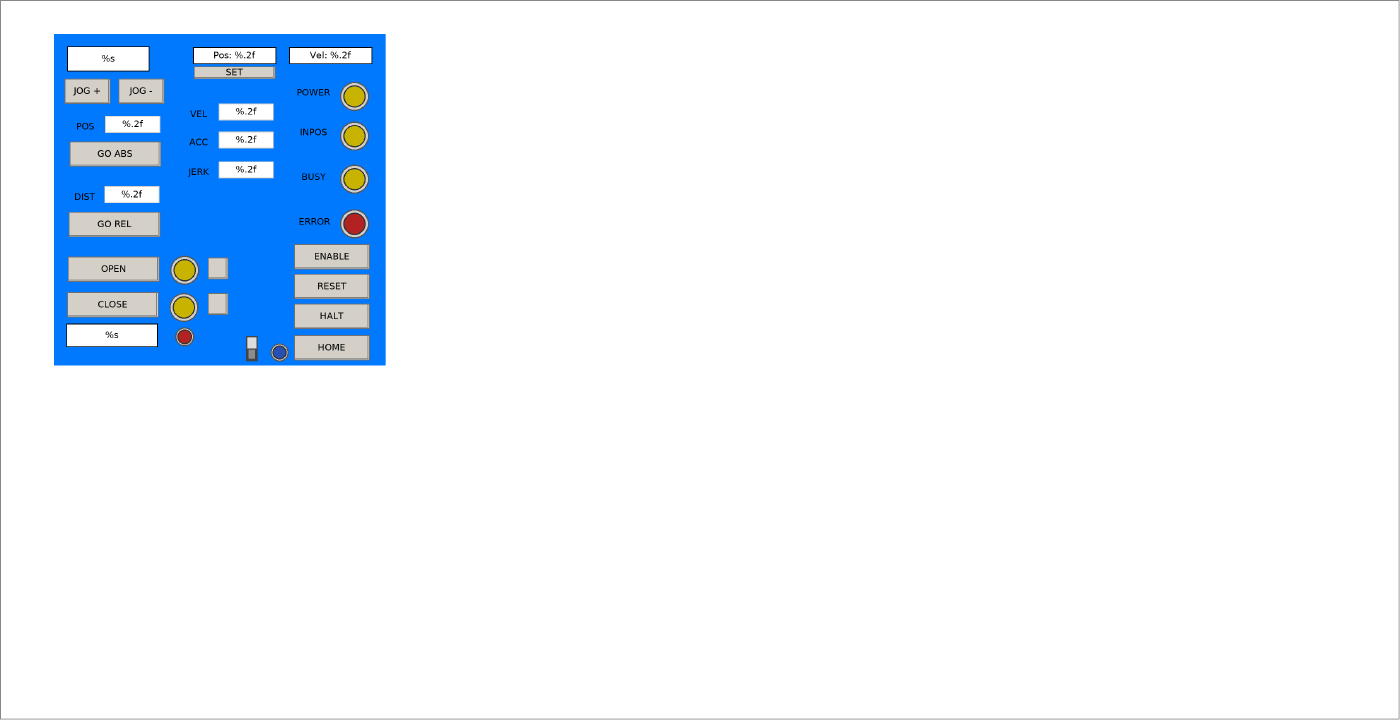
VISUALIZATION AXES_SCREEN  // 1690x870
    Frame (65,41 400x400)
        shows vAXIS(vAxis := MAIN_CONV)
END_VISUALIZATION

// ---- POUs/PISTONS/vPISTON.TcVIS
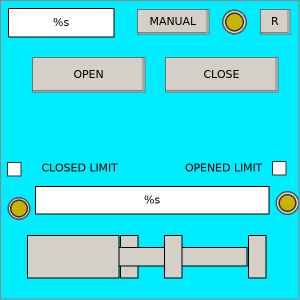
VISUALIZATION vPISTON  // 300x300
VAR_IN_OUT
	PIST1: FB_PISTON;
	
	
END_VAR
    Button (32,57 113x35), "OPEN"
        OnMouseDown: execute { PIST1.bOPEN_CMD:=TRUE; }
    Rectangle (35,186 234x28), "%s", text variable: PIST1.sSTATE
    Lamp1 (6,188 26x41), variable: PIST1.bCLOSED_LIMIT, style: Lamp-Lamp1-Yellow
    Label (30,153 99x30), "CLOSED LIMIT"
    Lamp1 (274,187 27x32), variable: PIST1.bOPEN_LIMIT, style: Lamp-Lamp1-Yellow
    Label (174,153 99x30), "OPENED LIMIT"
    Rectangle (8,8 106x29), "%s", text variable: PIST1.sNAME
    Button (165,57 113x35), "CLOSE"
        OnMouseDown: execute { PIST1.bOPEN_CMD:=FALSE; }
    Button (137,9 72x25), "MANUAL", colour toggle: PIST1.bLOCAL_MANUAL
        toggle PIST1.bLOCAL_MANUAL
    Lamp1 (219,8 31x28), variable: PIST1.bLOCAL_MANUAL, style: Lamp-Lamp1-Yellow
    Checkbox (5,154 34x30), variable: PIST1.bCLOSED_LIMIT
    Checkbox (270,153 34x30), variable: PIST1.bOPEN_LIMIT
    Button (260,9 30x25), "R", colour toggle: PIST1.bLOCAL_MANUAL
        tap PIST1.bLOCAL_RESET
    Rectangle (119,247 128x19), invisible if: NOT PIST1.bOPENED
    Rectangle (248,235 18x43), invisible if: NOT PIST1.bOPENED
    Rectangle (120,235 18x43), invisible if: NOT PIST1.bCLOSED
    Rectangle (78,247 92x19), invisible if: NOT PIST1.bBUSY
    Rectangle (164,235 18x43), invisible if: NOT PIST1.bBUSY
    Rectangle (27,235 92x43), colour toggle: PIST1.bERROR
END_VISUALIZATION

// ---- POUs/STATIONS/vFEEDER.TcVIS
